REGION Network 52: MB3 Code 4037 - REGOLAZ. BORDATRICE - PASSAGGIO 04 - COMBO
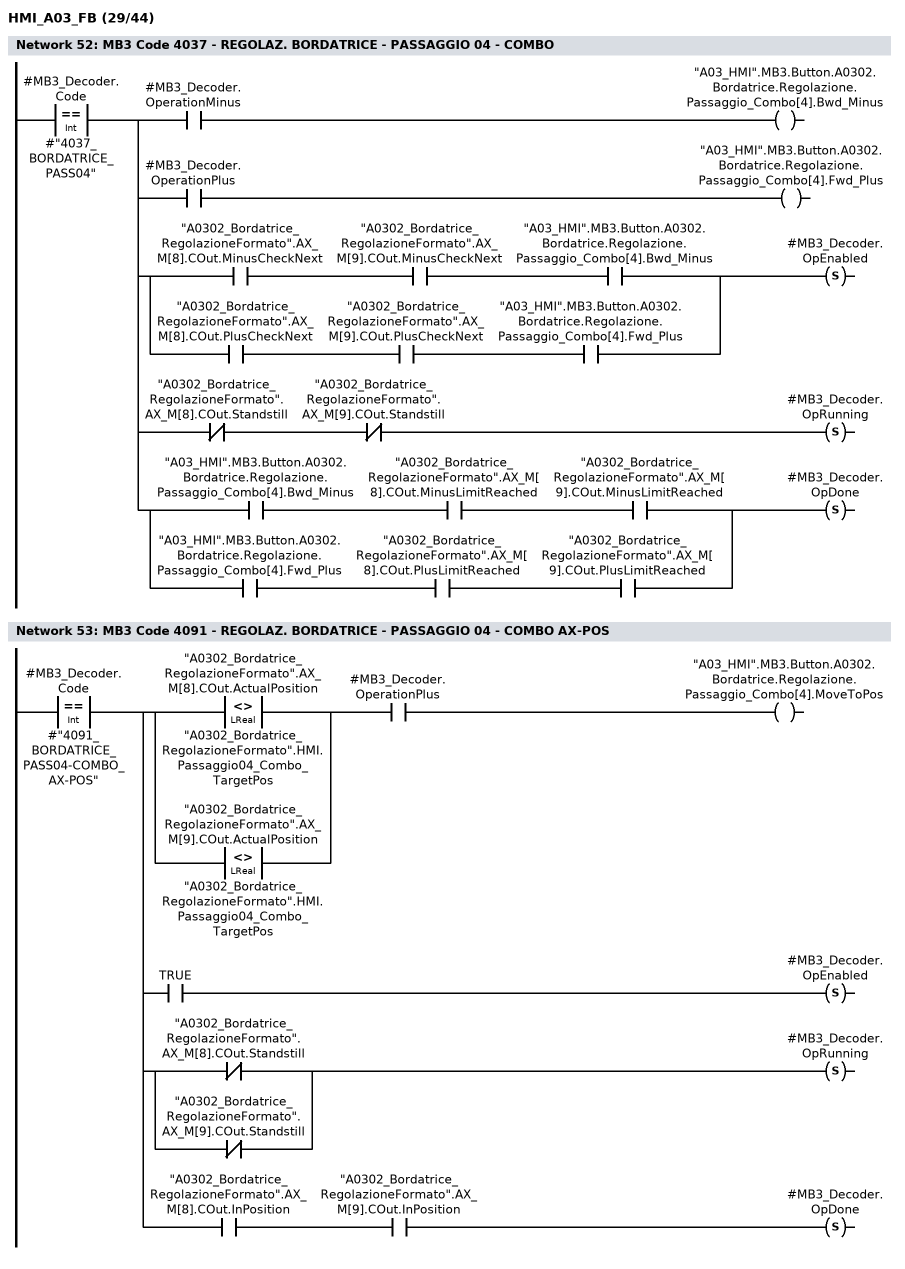
   RUNG wire#powerrail
      { S7_Templates := "SrcType := Int" } EQ_Contact(in1 := #MB3_Decoder.Code, in2 := #"4037_BORDATRICE_PASS04")
      wire#w1
      Contact( #MB3_Decoder.OperationMinus )
      Coil( "A03_HMI".MB3.Button.A0302.Bordatrice.Regolazione.Passaggio_Combo[4].Bwd_Minus )
   END_RUNG
   RUNG wire#w1
      Contact( #MB3_Decoder.OperationPlus )
      Coil( "A03_HMI".MB3.Button.A0302.Bordatrice.Regolazione.Passaggio_Combo[4].Fwd_Plus )
   END_RUNG
   RUNG wire#w1
      Contact( "A0302_Bordatrice_RegolazioneFormato".AX_M[8].COut.MinusCheckNext )
      Contact( "A0302_Bordatrice_RegolazioneFormato".AX_M[9].COut.MinusCheckNext )
      Contact( "A03_HMI".MB3.Button.A0302.Bordatrice.Regolazione.Passaggio_Combo[4].Bwd_Minus )
      wire#w2
      S_Coil( #MB3_Decoder.OpEnabled )
   END_RUNG
   RUNG wire#w1
      Contact( "A0302_Bordatrice_RegolazioneFormato".AX_M[8].COut.PlusCheckNext )
      Contact( "A0302_Bordatrice_RegolazioneFormato".AX_M[9].COut.PlusCheckNext )
      Contact( "A03_HMI".MB3.Button.A0302.Bordatrice.Regolazione.Passaggio_Combo[4].Fwd_Plus )
   END_RUNG wire#w2
   RUNG wire#w1
      I_Contact( "A0302_Bordatrice_RegolazioneFormato".AX_M[8].COut.Standstill )
      I_Contact( "A0302_Bordatrice_RegolazioneFormato".AX_M[9].COut.Standstill )
      S_Coil( #MB3_Decoder.OpRunning )
   END_RUNG
   RUNG wire#w1
      Contact( "A03_HMI".MB3.Button.A0302.Bordatrice.Regolazione.Passaggio_Combo[4].Bwd_Minus )
      Contact( "A0302_Bordatrice_RegolazioneFormato".AX_M[8].COut.MinusLimitReached )
      Contact( "A0302_Bordatrice_RegolazioneFormato".AX_M[9].COut.MinusLimitReached )
      wire#w3
      S_Coil( #MB3_Decoder.OpDone )
   END_RUNG
   RUNG wire#w1
      Contact( "A03_HMI".MB3.Button.A0302.Bordatrice.Regolazione.Passaggio_Combo[4].Fwd_Plus )
      Contact( "A0302_Bordatrice_RegolazioneFormato".AX_M[8].COut.PlusLimitReached )
      Contact( "A0302_Bordatrice_RegolazioneFormato".AX_M[9].COut.PlusLimitReached )
   END_RUNG wire#w3
   // the same network as SCL:
   #_w1 := #MB3_Decoder.Code = #"4037_BORDATRICE_PASS04";
   "A03_HMI".MB3.Button.A0302.Bordatrice.Regolazione.Passaggio_Combo[4].Bwd_Minus := #_w1 AND #MB3_Decoder.OperationMinus;
   "A03_HMI".MB3.Button.A0302.Bordatrice.Regolazione.Passaggio_Combo[4].Fwd_Plus := #_w1 AND #MB3_Decoder.OperationPlus;
   IF #_w1 AND (("A0302_Bordatrice_RegolazioneFormato".AX_M[8].COut.MinusCheckNext AND "A0302_Bordatrice_RegolazioneFormato".AX_M[9].COut.MinusCheckNext AND "A03_HMI".MB3.Button.A0302.Bordatrice.Regolazione.Passaggio_Combo[4].Bwd_Minus) OR ("A0302_Bordatrice_RegolazioneFormato".AX_M[8].COut.PlusCheckNext AND "A0302_Bordatrice_RegolazioneFormato".AX_M[9].COut.PlusCheckNext AND "A03_HMI".MB3.Button.A0302.Bordatrice.Regolazione.Passaggio_Combo[4].Fwd_Plus)) THEN
       #MB3_Decoder.OpEnabled := TRUE;
   END_IF;
   IF #_w1 AND NOT "A0302_Bordatrice_RegolazioneFormato".AX_M[8].COut.Standstill AND NOT "A0302_Bordatrice_RegolazioneFormato".AX_M[9].COut.Standstill THEN
       #MB3_Decoder.OpRunning := TRUE;
   END_IF;
   IF #_w1 AND (("A03_HMI".MB3.Button.A0302.Bordatrice.Regolazione.Passaggio_Combo[4].Bwd_Minus AND "A0302_Bordatrice_RegolazioneFormato".AX_M[8].COut.MinusLimitReached AND "A0302_Bordatrice_RegolazioneFormato".AX_M[9].COut.MinusLimitReached) OR ("A03_HMI".MB3.Button.A0302.Bordatrice.Regolazione.Passaggio_Combo[4].Fwd_Plus AND "A0302_Bordatrice_RegolazioneFormato".AX_M[8].COut.PlusLimitReached AND "A0302_Bordatrice_RegolazioneFormato".AX_M[9].COut.PlusLimitReached)) THEN
       #MB3_Decoder.OpDone := TRUE;
   END_IF;
END_REGION

REGION Network 53: MB3 Code 4091 - REGOLAZ. BORDATRICE - PASSAGGIO 04 - COMBO AX-POS
   RUNG wire#powerrail
      { S7_Templates := "SrcType := Int" } EQ_Contact(in1 := #MB3_Decoder.Code, in2 := #"4091_BORDATRICE_PASS04-COMBO_AX-POS")
      wire#w1
      { S7_Templates := "SrcType := LReal" } NE_Contact(in1 := "A0302_Bordatrice_RegolazioneFormato".AX_M[8].COut.ActualPosition, in2 := "A0302_Bordatrice_RegolazioneFormato".HMI.Passaggio04_Combo_TargetPos)
      wire#w2
      Contact( #MB3_Decoder.OperationPlus )
      Coil( "A03_HMI".MB3.Button.A0302.Bordatrice.Regolazione.Passaggio_Combo[4].MoveToPos )
   END_RUNG
   RUNG wire#w1
      { S7_Templates := "SrcType := LReal" } NE_Contact(in1 := "A0302_Bordatrice_RegolazioneFormato".AX_M[9].COut.ActualPosition, in2 := "A0302_Bordatrice_RegolazioneFormato".HMI.Passaggio04_Combo_TargetPos)
   END_RUNG wire#w2
   RUNG wire#w1
      Contact( TRUE )
      S_Coil( #MB3_Decoder.OpEnabled )
   END_RUNG
   RUNG wire#w1
      I_Contact( "A0302_Bordatrice_RegolazioneFormato".AX_M[8].COut.Standstill )
      wire#w3
      S_Coil( #MB3_Decoder.OpRunning )
   END_RUNG
   RUNG wire#w1
      I_Contact( "A0302_Bordatrice_RegolazioneFormato".AX_M[9].COut.Standstill )
   END_RUNG wire#w3
   RUNG wire#w1
      Contact( "A0302_Bordatrice_RegolazioneFormato".AX_M[8].COut.InPosition )
      Contact( "A0302_Bordatrice_RegolazioneFormato".AX_M[9].COut.InPosition )
      S_Coil( #MB3_Decoder.OpDone )
   END_RUNG
   // the same network as SCL:
   #_w1 := #MB3_Decoder.Code = #"4091_BORDATRICE_PASS04-COMBO_AX-POS";
   "A03_HMI".MB3.Button.A0302.Bordatrice.Regolazione.Passaggio_Combo[4].MoveToPos := #_w1 AND (("A0302_Bordatrice_RegolazioneFormato".AX_M[8].COut.ActualPosition <> "A0302_Bordatrice_RegolazioneFormato".HMI.Passaggio04_Combo_TargetPos) OR ("A0302_Bordatrice_RegolazioneFormato".AX_M[9].COut.ActualPosition <> "A0302_Bordatrice_RegolazioneFormato".HMI.Passaggio04_Combo_TargetPos)) AND #MB3_Decoder.OperationPlus;
   IF #_w1 AND TRUE THEN #MB3_Decoder.OpEnabled := TRUE; END_IF;
   IF #_w1 AND (NOT "A0302_Bordatrice_RegolazioneFormato".AX_M[8].COut.Standstill OR NOT "A0302_Bordatrice_RegolazioneFormato".AX_M[9].COut.Standstill) THEN
       #MB3_Decoder.OpRunning := TRUE;
   END_IF;
   IF #_w1 AND "A0302_Bordatrice_RegolazioneFormato".AX_M[8].COut.InPosition AND "A0302_Bordatrice_RegolazioneFormato".AX_M[9].COut.InPosition THEN
       #MB3_Decoder.OpDone := TRUE;
   END_IF;
END_REGION

REGION Network 54: MB3 Code 4086 - REGOLAZ. BORDATRICE - PASSAGGIO 04 - LATO-OP
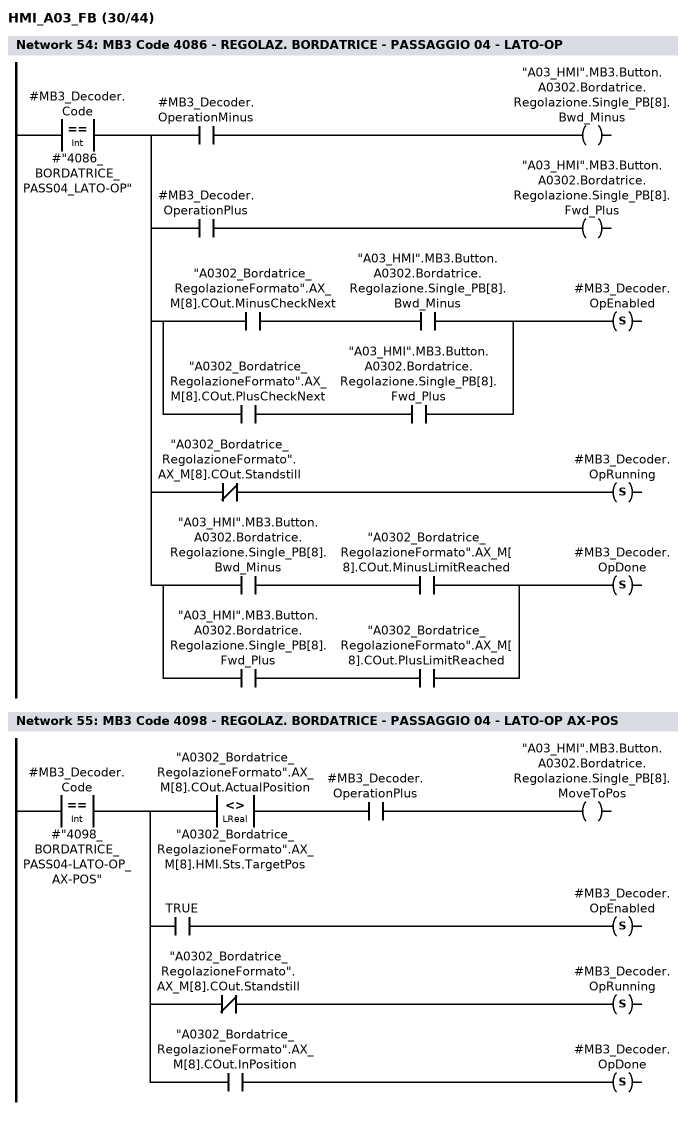
   RUNG wire#powerrail
      { S7_Templates := "SrcType := Int" } EQ_Contact(in1 := #MB3_Decoder.Code, in2 := #"4086_BORDATRICE_PASS04_LATO-OP")
      wire#w1
      Contact( #MB3_Decoder.OperationMinus )
      Coil( "A03_HMI".MB3.Button.A0302.Bordatrice.Regolazione.Single_PB[8].Bwd_Minus )
   END_RUNG
   RUNG wire#w1
      Contact( #MB3_Decoder.OperationPlus )
      Coil( "A03_HMI".MB3.Button.A0302.Bordatrice.Regolazione.Single_PB[8].Fwd_Plus )
   END_RUNG
   RUNG wire#w1
      Contact( "A0302_Bordatrice_RegolazioneFormato".AX_M[8].COut.MinusCheckNext )
      Contact( "A03_HMI".MB3.Button.A0302.Bordatrice.Regolazione.Single_PB[8].Bwd_Minus )
      wire#w2
      S_Coil( #MB3_Decoder.OpEnabled )
   END_RUNG
   RUNG wire#w1
      Contact( "A0302_Bordatrice_RegolazioneFormato".AX_M[8].COut.PlusCheckNext )
      Contact( "A03_HMI".MB3.Button.A0302.Bordatrice.Regolazione.Single_PB[8].Fwd_Plus )
   END_RUNG wire#w2
   RUNG wire#w1
      I_Contact( "A0302_Bordatrice_RegolazioneFormato".AX_M[8].COut.Standstill )
      S_Coil( #MB3_Decoder.OpRunning )
   END_RUNG
   RUNG wire#w1
      Contact( "A03_HMI".MB3.Button.A0302.Bordatrice.Regolazione.Single_PB[8].Bwd_Minus )
      Contact( "A0302_Bordatrice_RegolazioneFormato".AX_M[8].COut.MinusLimitReached )
      wire#w3
      S_Coil( #MB3_Decoder.OpDone )
   END_RUNG
   RUNG wire#w1
      Contact( "A03_HMI".MB3.Button.A0302.Bordatrice.Regolazione.Single_PB[8].Fwd_Plus )
      Contact( "A0302_Bordatrice_RegolazioneFormato".AX_M[8].COut.PlusLimitReached )
   END_RUNG wire#w3
   // the same network as SCL:
   #_w1 := #MB3_Decoder.Code = #"4086_BORDATRICE_PASS04_LATO-OP";
   "A03_HMI".MB3.Button.A0302.Bordatrice.Regolazione.Single_PB[8].Bwd_Minus := #_w1 AND #MB3_Decoder.OperationMinus;
   "A03_HMI".MB3.Button.A0302.Bordatrice.Regolazione.Single_PB[8].Fwd_Plus := #_w1 AND #MB3_Decoder.OperationPlus;
   IF #_w1 AND (("A0302_Bordatrice_RegolazioneFormato".AX_M[8].COut.MinusCheckNext AND "A03_HMI".MB3.Button.A0302.Bordatrice.Regolazione.Single_PB[8].Bwd_Minus) OR ("A0302_Bordatrice_RegolazioneFormato".AX_M[8].COut.PlusCheckNext AND "A03_HMI".MB3.Button.A0302.Bordatrice.Regolazione.Single_PB[8].Fwd_Plus)) THEN
       #MB3_Decoder.OpEnabled := TRUE;
   END_IF;
   IF #_w1 AND NOT "A0302_Bordatrice_RegolazioneFormato".AX_M[8].COut.Standstill THEN
       #MB3_Decoder.OpRunning := TRUE;
   END_IF;
   IF #_w1 AND (("A03_HMI".MB3.Button.A0302.Bordatrice.Regolazione.Single_PB[8].Bwd_Minus AND "A0302_Bordatrice_RegolazioneFormato".AX_M[8].COut.MinusLimitReached) OR ("A03_HMI".MB3.Button.A0302.Bordatrice.Regolazione.Single_PB[8].Fwd_Plus AND "A0302_Bordatrice_RegolazioneFormato".AX_M[8].COut.PlusLimitReached)) THEN
       #MB3_Decoder.OpDone := TRUE;
   END_IF;
END_REGION

REGION Network 55: MB3 Code 4098 - REGOLAZ. BORDATRICE - PASSAGGIO 04 - LATO-OP AX-POS
   RUNG wire#powerrail
      { S7_Templates := "SrcType := Int" } EQ_Contact(in1 := #MB3_Decoder.Code, in2 := #"4098_BORDATRICE_PASS04-LATO-OP_AX-POS")
      wire#w1
      { S7_Templates := "SrcType := LReal" } NE_Contact(in1 := "A0302_Bordatrice_RegolazioneFormato".AX_M[8].COut.ActualPosition, in2 := "A0302_Bordatrice_RegolazioneFormato".AX_M[8].HMI.Sts.TargetPos)
      Contact( #MB3_Decoder.OperationPlus )
      Coil( "A03_HMI".MB3.Button.A0302.Bordatrice.Regolazione.Single_PB[8].MoveToPos )
   END_RUNG
   RUNG wire#w1
      Contact( TRUE )
      S_Coil( #MB3_Decoder.OpEnabled )
   END_RUNG
   RUNG wire#w1
      I_Contact( "A0302_Bordatrice_RegolazioneFormato".AX_M[8].COut.Standstill )
      S_Coil( #MB3_Decoder.OpRunning )
   END_RUNG
   RUNG wire#w1
      Contact( "A0302_Bordatrice_RegolazioneFormato".AX_M[8].COut.InPosition )
      S_Coil( #MB3_Decoder.OpDone )
   END_RUNG
   // the same network as SCL:
   #_w1 := #MB3_Decoder.Code = #"4098_BORDATRICE_PASS04-LATO-OP_AX-POS";
   "A03_HMI".MB3.Button.A0302.Bordatrice.Regolazione.Single_PB[8].MoveToPos := #_w1 AND ("A0302_Bordatrice_RegolazioneFormato".AX_M[8].COut.ActualPosition <> "A0302_Bordatrice_RegolazioneFormato".AX_M[8].HMI.Sts.TargetPos) AND #MB3_Decoder.OperationPlus;
   IF #_w1 AND TRUE THEN #MB3_Decoder.OpEnabled := TRUE; END_IF;
   IF #_w1 AND NOT "A0302_Bordatrice_RegolazioneFormato".AX_M[8].COut.Standstill THEN
       #MB3_Decoder.OpRunning := TRUE;
   END_IF;
   IF #_w1 AND "A0302_Bordatrice_RegolazioneFormato".AX_M[8].COut.InPosition THEN
       #MB3_Decoder.OpDone := TRUE;
   END_IF;
END_REGION

REGION Network 56: MB3 Code 4087 - REGOLAZ. BORDATRICE - PASSAGGIO 04 - LATO-MOT
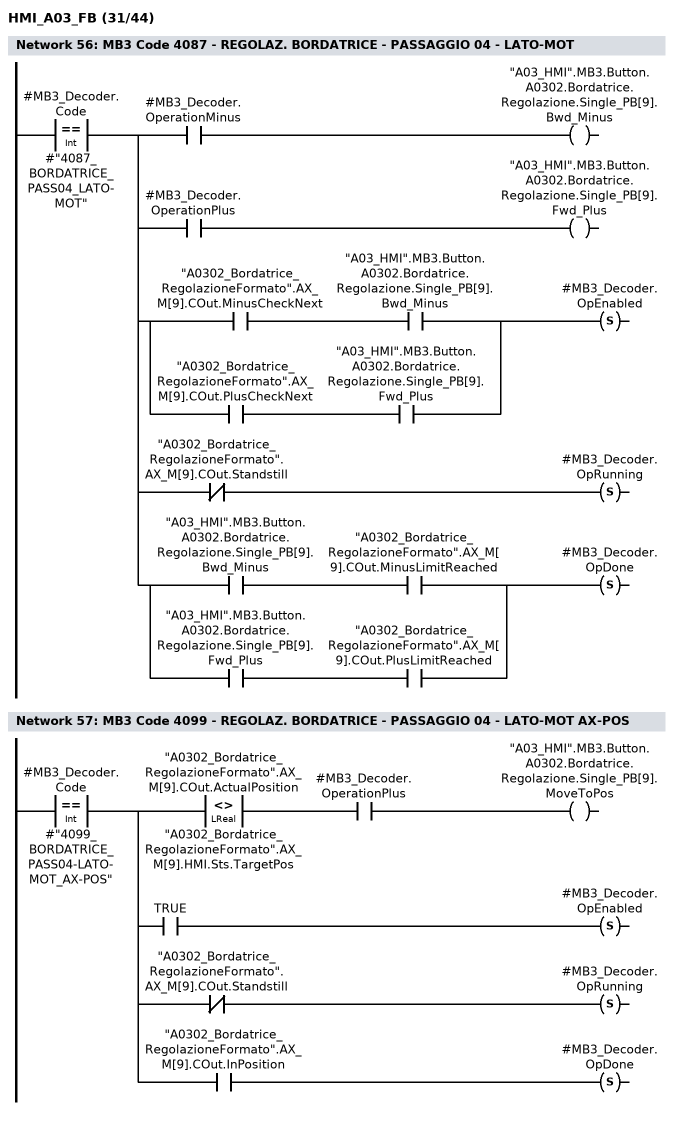
   RUNG wire#powerrail
      { S7_Templates := "SrcType := Int" } EQ_Contact(in1 := #MB3_Decoder.Code, in2 := #"4087_BORDATRICE_PASS04_LATO-MOT")
      wire#w1
      Contact( #MB3_Decoder.OperationMinus )
      Coil( "A03_HMI".MB3.Button.A0302.Bordatrice.Regolazione.Single_PB[9].Bwd_Minus )
   END_RUNG
   RUNG wire#w1
      Contact( #MB3_Decoder.OperationPlus )
      Coil( "A03_HMI".MB3.Button.A0302.Bordatrice.Regolazione.Single_PB[9].Fwd_Plus )
   END_RUNG
   RUNG wire#w1
      Contact( "A0302_Bordatrice_RegolazioneFormato".AX_M[9].COut.MinusCheckNext )
      Contact( "A03_HMI".MB3.Button.A0302.Bordatrice.Regolazione.Single_PB[9].Bwd_Minus )
      wire#w2
      S_Coil( #MB3_Decoder.OpEnabled )
   END_RUNG
   RUNG wire#w1
      Contact( "A0302_Bordatrice_RegolazioneFormato".AX_M[9].COut.PlusCheckNext )
      Contact( "A03_HMI".MB3.Button.A0302.Bordatrice.Regolazione.Single_PB[9].Fwd_Plus )
   END_RUNG wire#w2
   RUNG wire#w1
      I_Contact( "A0302_Bordatrice_RegolazioneFormato".AX_M[9].COut.Standstill )
      S_Coil( #MB3_Decoder.OpRunning )
   END_RUNG
   RUNG wire#w1
      Contact( "A03_HMI".MB3.Button.A0302.Bordatrice.Regolazione.Single_PB[9].Bwd_Minus )
      Contact( "A0302_Bordatrice_RegolazioneFormato".AX_M[9].COut.MinusLimitReached )
      wire#w3
      S_Coil( #MB3_Decoder.OpDone )
   END_RUNG
   RUNG wire#w1
      Contact( "A03_HMI".MB3.Button.A0302.Bordatrice.Regolazione.Single_PB[9].Fwd_Plus )
      Contact( "A0302_Bordatrice_RegolazioneFormato".AX_M[9].COut.PlusLimitReached )
   END_RUNG wire#w3
   // the same network as SCL:
   #_w1 := #MB3_Decoder.Code = #"4087_BORDATRICE_PASS04_LATO-MOT";
   "A03_HMI".MB3.Button.A0302.Bordatrice.Regolazione.Single_PB[9].Bwd_Minus := #_w1 AND #MB3_Decoder.OperationMinus;
   "A03_HMI".MB3.Button.A0302.Bordatrice.Regolazione.Single_PB[9].Fwd_Plus := #_w1 AND #MB3_Decoder.OperationPlus;
   IF #_w1 AND (("A0302_Bordatrice_RegolazioneFormato".AX_M[9].COut.MinusCheckNext AND "A03_HMI".MB3.Button.A0302.Bordatrice.Regolazione.Single_PB[9].Bwd_Minus) OR ("A0302_Bordatrice_RegolazioneFormato".AX_M[9].COut.PlusCheckNext AND "A03_HMI".MB3.Button.A0302.Bordatrice.Regolazione.Single_PB[9].Fwd_Plus)) THEN
       #MB3_Decoder.OpEnabled := TRUE;
   END_IF;
   IF #_w1 AND NOT "A0302_Bordatrice_RegolazioneFormato".AX_M[9].COut.Standstill THEN
       #MB3_Decoder.OpRunning := TRUE;
   END_IF;
   IF #_w1 AND (("A03_HMI".MB3.Button.A0302.Bordatrice.Regolazione.Single_PB[9].Bwd_Minus AND "A0302_Bordatrice_RegolazioneFormato".AX_M[9].COut.MinusLimitReached) OR ("A03_HMI".MB3.Button.A0302.Bordatrice.Regolazione.Single_PB[9].Fwd_Plus AND "A0302_Bordatrice_RegolazioneFormato".AX_M[9].COut.PlusLimitReached)) THEN
       #MB3_Decoder.OpDone := TRUE;
   END_IF;
END_REGION

REGION Network 57: MB3 Code 4099 - REGOLAZ. BORDATRICE - PASSAGGIO 04 - LATO-MOT AX-POS
   RUNG wire#powerrail
      { S7_Templates := "SrcType := Int" } EQ_Contact(in1 := #MB3_Decoder.Code, in2 := #"4099_BORDATRICE_PASS04-LATO-MOT_AX-POS")
      wire#w1
      { S7_Templates := "SrcType := LReal" } NE_Contact(in1 := "A0302_Bordatrice_RegolazioneFormato".AX_M[9].COut.ActualPosition, in2 := "A0302_Bordatrice_RegolazioneFormato".AX_M[9].HMI.Sts.TargetPos)
      Contact( #MB3_Decoder.OperationPlus )
      Coil( "A03_HMI".MB3.Button.A0302.Bordatrice.Regolazione.Single_PB[9].MoveToPos )
   END_RUNG
   RUNG wire#w1
      Contact( TRUE )
      S_Coil( #MB3_Decoder.OpEnabled )
   END_RUNG
   RUNG wire#w1
      I_Contact( "A0302_Bordatrice_RegolazioneFormato".AX_M[9].COut.Standstill )
      S_Coil( #MB3_Decoder.OpRunning )
   END_RUNG
   RUNG wire#w1
      Contact( "A0302_Bordatrice_RegolazioneFormato".AX_M[9].COut.InPosition )
      S_Coil( #MB3_Decoder.OpDone )
   END_RUNG
   // the same network as SCL:
   #_w1 := #MB3_Decoder.Code = #"4099_BORDATRICE_PASS04-LATO-MOT_AX-POS";
   "A03_HMI".MB3.Button.A0302.Bordatrice.Regolazione.Single_PB[9].MoveToPos := #_w1 AND ("A0302_Bordatrice_RegolazioneFormato".AX_M[9].COut.ActualPosition <> "A0302_Bordatrice_RegolazioneFormato".AX_M[9].HMI.Sts.TargetPos) AND #MB3_Decoder.OperationPlus;
   IF #_w1 AND TRUE THEN #MB3_Decoder.OpEnabled := TRUE; END_IF;
   IF #_w1 AND NOT "A0302_Bordatrice_RegolazioneFormato".AX_M[9].COut.Standstill THEN
       #MB3_Decoder.OpRunning := TRUE;
   END_IF;
   IF #_w1 AND "A0302_Bordatrice_RegolazioneFormato".AX_M[9].COut.InPosition THEN
       #MB3_Decoder.OpDone := TRUE;
   END_IF;
END_REGION

REGION Network 58: MB3 Code 4041- CENTARTORI - OP
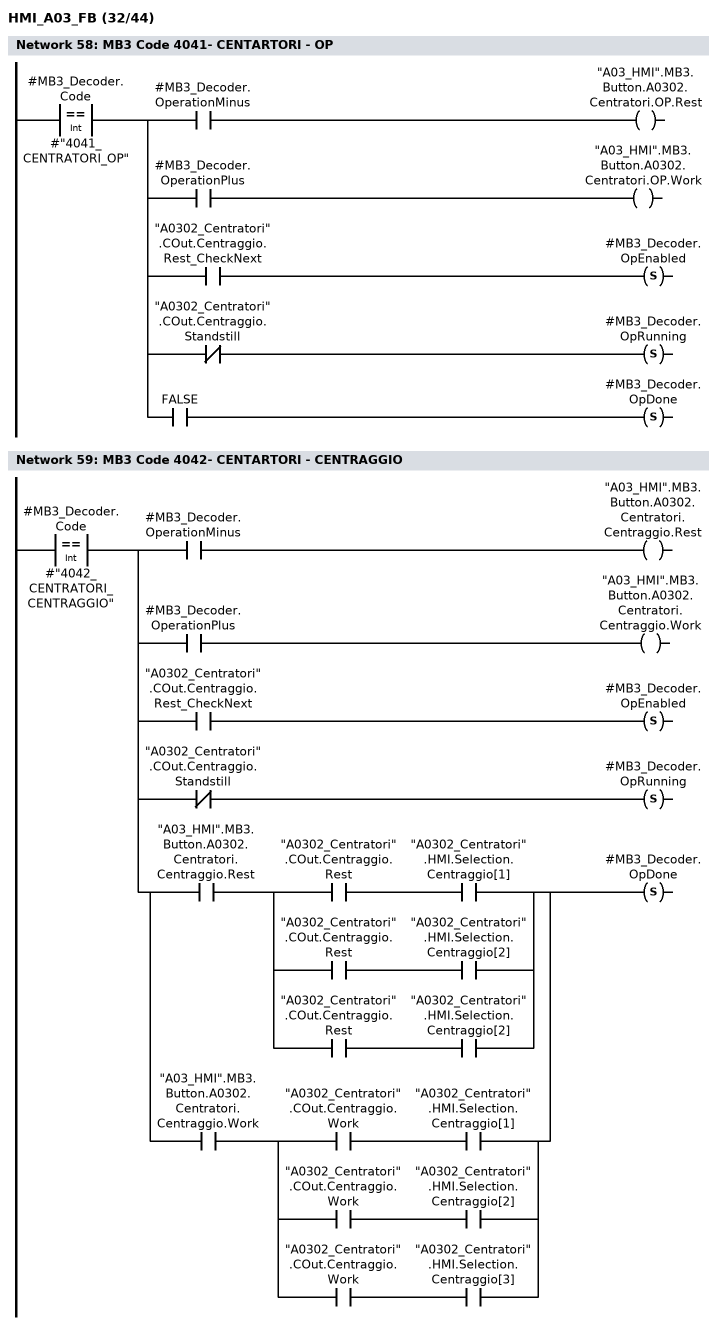
   RUNG wire#powerrail
      { S7_Templates := "SrcType := Int" } EQ_Contact(in1 := #MB3_Decoder.Code, in2 := #"4041_CENTRATORI_OP")
      wire#w1
      Contact( #MB3_Decoder.OperationMinus )
      Coil( "A03_HMI".MB3.Button.A0302.Centratori.OP.Rest )
   END_RUNG
   RUNG wire#w1
      Contact( #MB3_Decoder.OperationPlus )
      Coil( "A03_HMI".MB3.Button.A0302.Centratori.OP.Work )
   END_RUNG
   RUNG wire#w1
      Contact( "A0302_Centratori".COut.Centraggio.Rest_CheckNext )
      S_Coil( #MB3_Decoder.OpEnabled )
   END_RUNG
   RUNG wire#w1
      I_Contact( "A0302_Centratori".COut.Centraggio.Standstill )
      S_Coil( #MB3_Decoder.OpRunning )
   END_RUNG
   RUNG wire#w1
      Contact( FALSE )
      S_Coil( #MB3_Decoder.OpDone )
   END_RUNG
   // the same network as SCL:
   #_w1 := #MB3_Decoder.Code = #"4041_CENTRATORI_OP";
   "A03_HMI".MB3.Button.A0302.Centratori.OP.Rest := #_w1 AND #MB3_Decoder.OperationMinus;
   "A03_HMI".MB3.Button.A0302.Centratori.OP.Work := #_w1 AND #MB3_Decoder.OperationPlus;
   IF #_w1 AND "A0302_Centratori".COut.Centraggio.Rest_CheckNext THEN #MB3_Decoder.OpEnabled := TRUE; END_IF;
   IF #_w1 AND NOT "A0302_Centratori".COut.Centraggio.Standstill THEN #MB3_Decoder.OpRunning := TRUE; END_IF;
   IF #_w1 AND FALSE THEN #MB3_Decoder.OpDone := TRUE; END_IF;
END_REGION

REGION Network 59: MB3 Code 4042- CENTARTORI - CENTRAGGIO
   RUNG wire#powerrail
      { S7_Templates := "SrcType := Int" } EQ_Contact(in1 := #MB3_Decoder.Code, in2 := #"4042_CENTRATORI_CENTRAGGIO")
      wire#w1
      Contact( #MB3_Decoder.OperationMinus )
      Coil( "A03_HMI".MB3.Button.A0302.Centratori.Centraggio.Rest )
   END_RUNG
   RUNG wire#w1
      Contact( #MB3_Decoder.OperationPlus )
      Coil( "A03_HMI".MB3.Button.A0302.Centratori.Centraggio.Work )
   END_RUNG
   RUNG wire#w1
      Contact( "A0302_Centratori".COut.Centraggio.Rest_CheckNext )
      S_Coil( #MB3_Decoder.OpEnabled )
   END_RUNG
   RUNG wire#w1
      I_Contact( "A0302_Centratori".COut.Centraggio.Standstill )
      S_Coil( #MB3_Decoder.OpRunning )
   END_RUNG
   RUNG wire#w1
      Contact( "A03_HMI".MB3.Button.A0302.Centratori.Centraggio.Rest )
      wire#w2
      Contact( "A0302_Centratori".COut.Centraggio.Rest )
      Contact( "A0302_Centratori".HMI.Selection.Centraggio[1] )
      wire#w3
      S_Coil( #MB3_Decoder.OpDone )
   END_RUNG
   RUNG wire#w2
      Contact( "A0302_Centratori".COut.Centraggio.Rest )
      Contact( "A0302_Centratori".HMI.Selection.Centraggio[2] )
   END_RUNG wire#w3
   RUNG wire#w2
      Contact( "A0302_Centratori".COut.Centraggio.Rest )
      Contact( "A0302_Centratori".HMI.Selection.Centraggio[2] )
   END_RUNG wire#w3
   RUNG wire#w1
      Contact( "A03_HMI".MB3.Button.A0302.Centratori.Centraggio.Work )
      wire#w4
      Contact( "A0302_Centratori".COut.Centraggio.Work )
      Contact( "A0302_Centratori".HMI.Selection.Centraggio[1] )
   END_RUNG wire#w3
   RUNG wire#w4
      Contact( "A0302_Centratori".COut.Centraggio.Work )
      Contact( "A0302_Centratori".HMI.Selection.Centraggio[2] )
   END_RUNG wire#w3
   RUNG wire#w4
      Contact( "A0302_Centratori".COut.Centraggio.Work )
      Contact( "A0302_Centratori".HMI.Selection.Centraggio[3] )
   END_RUNG wire#w3
   // the same network as SCL:
   #_w1 := #MB3_Decoder.Code = #"4042_CENTRATORI_CENTRAGGIO";
   "A03_HMI".MB3.Button.A0302.Centratori.Centraggio.Rest := #_w1 AND #MB3_Decoder.OperationMinus;
   "A03_HMI".MB3.Button.A0302.Centratori.Centraggio.Work := #_w1 AND #MB3_Decoder.OperationPlus;
   IF #_w1 AND "A0302_Centratori".COut.Centraggio.Rest_CheckNext THEN #MB3_Decoder.OpEnabled := TRUE; END_IF;
   IF #_w1 AND NOT "A0302_Centratori".COut.Centraggio.Standstill THEN #MB3_Decoder.OpRunning := TRUE; END_IF;
   IF #_w1 AND (("A03_HMI".MB3.Button.A0302.Centratori.Centraggio.Rest AND (("A0302_Centratori".COut.Centraggio.Rest AND "A0302_Centratori".HMI.Selection.Centraggio[1]) OR ("A0302_Centratori".COut.Centraggio.Rest AND "A0302_Centratori".HMI.Selection.Centraggio[2]) OR ("A0302_Centratori".COut.Centraggio.Rest AND "A0302_Centratori".HMI.Selection.Centraggio[2]))) OR ("A03_HMI".MB3.Button.A0302.Centratori.Centraggio.Work AND (("A0302_Centratori".COut.Centraggio.Work AND "A0302_Centratori".HMI.Selection.Centraggio[1]) OR ("A0302_Centratori".COut.Centraggio.Work AND "A0302_Centratori".HMI.Selection.Centraggio[2]) OR ("A0302_Centratori".COut.Centraggio.Work AND "A0302_Centratori".HMI.Selection.Centraggio[3])))) THEN
       #MB3_Decoder.OpDone := TRUE;
   END_IF;
END_REGION

REGION Network 60: MB3 Code 4043- CENTARTORI - SOLLEVAMENTO
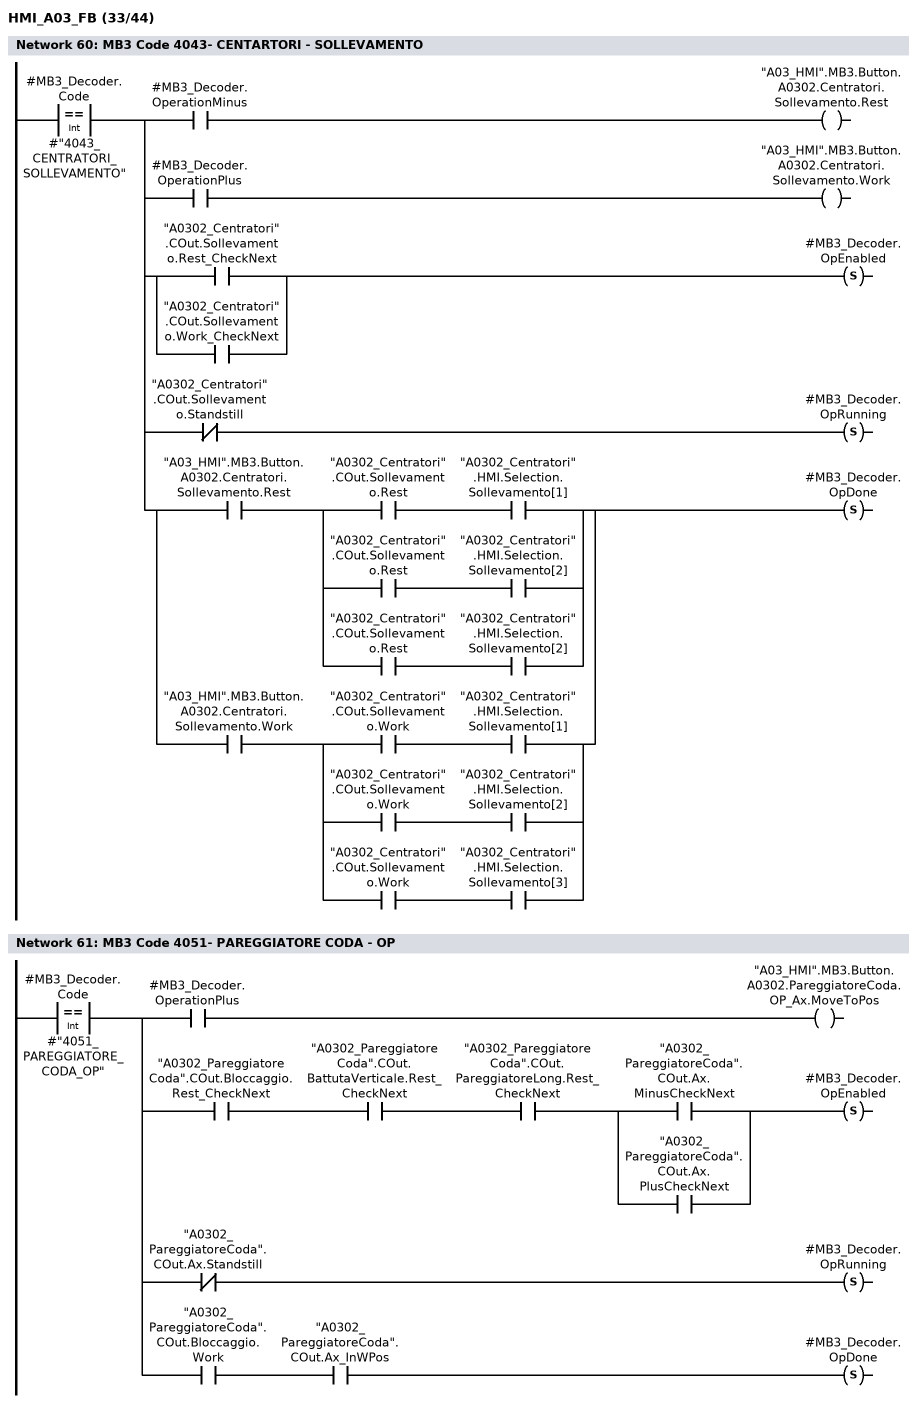
   RUNG wire#powerrail
      { S7_Templates := "SrcType := Int" } EQ_Contact(in1 := #MB3_Decoder.Code, in2 := #"4043_CENTRATORI_SOLLEVAMENTO")
      wire#w1
      Contact( #MB3_Decoder.OperationMinus )
      Coil( "A03_HMI".MB3.Button.A0302.Centratori.Sollevamento.Rest )
   END_RUNG
   RUNG wire#w1
      Contact( #MB3_Decoder.OperationPlus )
      Coil( "A03_HMI".MB3.Button.A0302.Centratori.Sollevamento.Work )
   END_RUNG
   RUNG wire#w1
      Contact( "A0302_Centratori".COut.Sollevamento.Rest_CheckNext )
      wire#w2
      S_Coil( #MB3_Decoder.OpEnabled )
   END_RUNG
   RUNG wire#w1
      Contact( "A0302_Centratori".COut.Sollevamento.Work_CheckNext )
   END_RUNG wire#w2
   RUNG wire#w1
      I_Contact( "A0302_Centratori".COut.Sollevamento.Standstill )
      S_Coil( #MB3_Decoder.OpRunning )
   END_RUNG
   RUNG wire#w1
      Contact( "A03_HMI".MB3.Button.A0302.Centratori.Sollevamento.Rest )
      wire#w3
      Contact( "A0302_Centratori".COut.Sollevamento.Rest )
      Contact( "A0302_Centratori".HMI.Selection.Sollevamento[1] )
      wire#w4
      S_Coil( #MB3_Decoder.OpDone )
   END_RUNG
   RUNG wire#w3
      Contact( "A0302_Centratori".COut.Sollevamento.Rest )
      Contact( "A0302_Centratori".HMI.Selection.Sollevamento[2] )
   END_RUNG wire#w4
   RUNG wire#w3
      Contact( "A0302_Centratori".COut.Sollevamento.Rest )
      Contact( "A0302_Centratori".HMI.Selection.Sollevamento[2] )
   END_RUNG wire#w4
   RUNG wire#w1
      Contact( "A03_HMI".MB3.Button.A0302.Centratori.Sollevamento.Work )
      wire#w5
      Contact( "A0302_Centratori".COut.Sollevamento.Work )
      Contact( "A0302_Centratori".HMI.Selection.Sollevamento[1] )
   END_RUNG wire#w4
   RUNG wire#w5
      Contact( "A0302_Centratori".COut.Sollevamento.Work )
      Contact( "A0302_Centratori".HMI.Selection.Sollevamento[2] )
   END_RUNG wire#w4
   RUNG wire#w5
      Contact( "A0302_Centratori".COut.Sollevamento.Work )
      Contact( "A0302_Centratori".HMI.Selection.Sollevamento[3] )
   END_RUNG wire#w4
   // the same network as SCL:
   #_w1 := #MB3_Decoder.Code = #"4043_CENTRATORI_SOLLEVAMENTO";
   "A03_HMI".MB3.Button.A0302.Centratori.Sollevamento.Rest := #_w1 AND #MB3_Decoder.OperationMinus;
   "A03_HMI".MB3.Button.A0302.Centratori.Sollevamento.Work := #_w1 AND #MB3_Decoder.OperationPlus;
   IF #_w1 AND ("A0302_Centratori".COut.Sollevamento.Rest_CheckNext OR "A0302_Centratori".COut.Sollevamento.Work_CheckNext) THEN
       #MB3_Decoder.OpEnabled := TRUE;
   END_IF;
   IF #_w1 AND NOT "A0302_Centratori".COut.Sollevamento.Standstill THEN
       #MB3_Decoder.OpRunning := TRUE;
   END_IF;
   IF #_w1 AND (("A03_HMI".MB3.Button.A0302.Centratori.Sollevamento.Rest AND (("A0302_Centratori".COut.Sollevamento.Rest AND "A0302_Centratori".HMI.Selection.Sollevamento[1]) OR ("A0302_Centratori".COut.Sollevamento.Rest AND "A0302_Centratori".HMI.Selection.Sollevamento[2]) OR ("A0302_Centratori".COut.Sollevamento.Rest AND "A0302_Centratori".HMI.Selection.Sollevamento[2]))) OR ("A03_HMI".MB3.Button.A0302.Centratori.Sollevamento.Work AND (("A0302_Centratori".COut.Sollevamento.Work AND "A0302_Centratori".HMI.Selection.Sollevamento[1]) OR ("A0302_Centratori".COut.Sollevamento.Work AND "A0302_Centratori".HMI.Selection.Sollevamento[2]) OR ("A0302_Centratori".COut.Sollevamento.Work AND "A0302_Centratori".HMI.Selection.Sollevamento[3])))) THEN
       #MB3_Decoder.OpDone := TRUE;
   END_IF;
END_REGION

REGION Network 61: MB3 Code 4051- PAREGGIATORE CODA - OP
   RUNG wire#powerrail
      { S7_Templates := "SrcType := Int" } EQ_Contact(in1 := #MB3_Decoder.Code, in2 := #"4051_PAREGGIATORE_CODA_OP")
      wire#w1
      Contact( #MB3_Decoder.OperationPlus )
      Coil( "A03_HMI".MB3.Button.A0302.PareggiatoreCoda.OP_Ax.MoveToPos )
   END_RUNG
   RUNG wire#w1
      Contact( "A0302_PareggiatoreCoda".COut.Bloccaggio.Rest_CheckNext )
      Contact( "A0302_PareggiatoreCoda".COut.BattutaVerticale.Rest_CheckNext )
      Contact( "A0302_PareggiatoreCoda".COut.PareggiatoreLong.Rest_CheckNext )
      wire#w2
      Contact( "A0302_PareggiatoreCoda".COut.Ax.MinusCheckNext )
      wire#w3
      S_Coil( #MB3_Decoder.OpEnabled )
   END_RUNG
   RUNG wire#w2
      Contact( "A0302_PareggiatoreCoda".COut.Ax.PlusCheckNext )
   END_RUNG wire#w3
   RUNG wire#w1
      I_Contact( "A0302_PareggiatoreCoda".COut.Ax.Standstill )
      S_Coil( #MB3_Decoder.OpRunning )
   END_RUNG
   RUNG wire#w1
      Contact( "A0302_PareggiatoreCoda".COut.Bloccaggio.Work )
      Contact( "A0302_PareggiatoreCoda".COut.Ax_InWPos )
      S_Coil( #MB3_Decoder.OpDone )
   END_RUNG
   // the same network as SCL:
   #_w1 := #MB3_Decoder.Code = #"4051_PAREGGIATORE_CODA_OP";
   "A03_HMI".MB3.Button.A0302.PareggiatoreCoda.OP_Ax.MoveToPos := #_w1 AND #MB3_Decoder.OperationPlus;
   IF #_w1 AND "A0302_PareggiatoreCoda".COut.Bloccaggio.Rest_CheckNext AND "A0302_PareggiatoreCoda".COut.BattutaVerticale.Rest_CheckNext AND "A0302_PareggiatoreCoda".COut.PareggiatoreLong.Rest_CheckNext AND ("A0302_PareggiatoreCoda".COut.Ax.MinusCheckNext OR "A0302_PareggiatoreCoda".COut.Ax.PlusCheckNext) THEN
       #MB3_Decoder.OpEnabled := TRUE;
   END_IF;
   IF #_w1 AND NOT "A0302_PareggiatoreCoda".COut.Ax.Standstill THEN #MB3_Decoder.OpRunning := TRUE; END_IF;
   IF #_w1 AND "A0302_PareggiatoreCoda".COut.Bloccaggio.Work AND "A0302_PareggiatoreCoda".COut.Ax_InWPos THEN
       #MB3_Decoder.OpDone := TRUE;
   END_IF;
END_REGION

REGION Network 62: MB3 Code 4052 - PAREGGIATORE CODA -AX
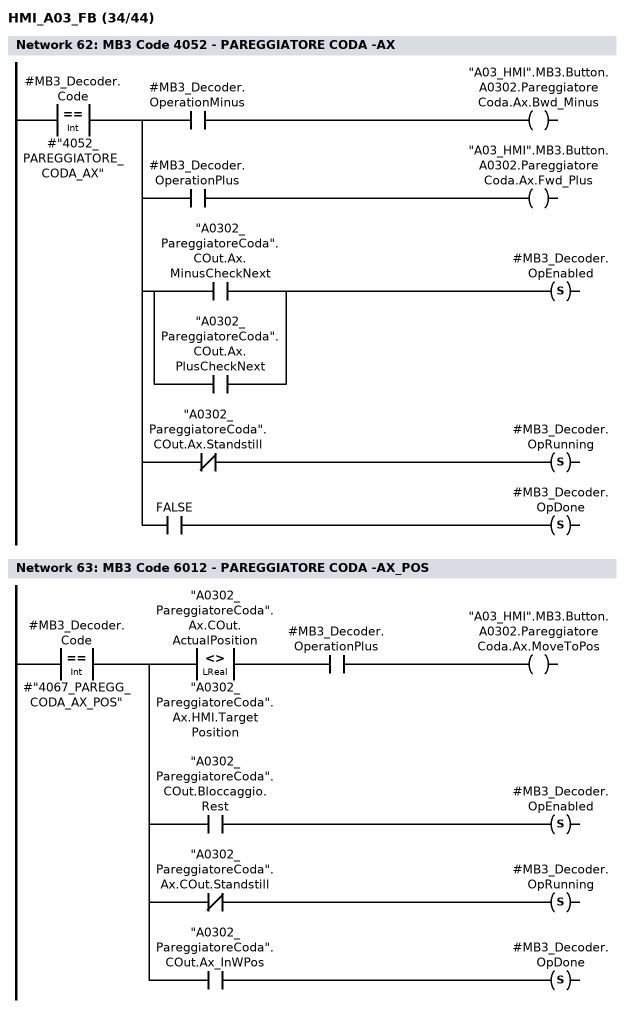
   RUNG wire#powerrail
      { S7_Templates := "SrcType := Int" } EQ_Contact(in1 := #MB3_Decoder.Code, in2 := #"4052_PAREGGIATORE_CODA_AX")
      wire#w1
      Contact( #MB3_Decoder.OperationMinus )
      Coil( "A03_HMI".MB3.Button.A0302.PareggiatoreCoda.Ax.Bwd_Minus )
   END_RUNG
   RUNG wire#w1
      Contact( #MB3_Decoder.OperationPlus )
      Coil( "A03_HMI".MB3.Button.A0302.PareggiatoreCoda.Ax.Fwd_Plus )
   END_RUNG
   RUNG wire#w1
      Contact( "A0302_PareggiatoreCoda".COut.Ax.MinusCheckNext )
      wire#w2
      S_Coil( #MB3_Decoder.OpEnabled )
   END_RUNG
   RUNG wire#w1
      Contact( "A0302_PareggiatoreCoda".COut.Ax.PlusCheckNext )
   END_RUNG wire#w2
   RUNG wire#w1
      I_Contact( "A0302_PareggiatoreCoda".COut.Ax.Standstill )
      S_Coil( #MB3_Decoder.OpRunning )
   END_RUNG
   RUNG wire#w1
      Contact( FALSE )
      S_Coil( #MB3_Decoder.OpDone )
   END_RUNG
   // the same network as SCL:
   #_w1 := #MB3_Decoder.Code = #"4052_PAREGGIATORE_CODA_AX";
   "A03_HMI".MB3.Button.A0302.PareggiatoreCoda.Ax.Bwd_Minus := #_w1 AND #MB3_Decoder.OperationMinus;
   "A03_HMI".MB3.Button.A0302.PareggiatoreCoda.Ax.Fwd_Plus := #_w1 AND #MB3_Decoder.OperationPlus;
   IF #_w1 AND ("A0302_PareggiatoreCoda".COut.Ax.MinusCheckNext OR "A0302_PareggiatoreCoda".COut.Ax.PlusCheckNext) THEN
       #MB3_Decoder.OpEnabled := TRUE;
   END_IF;
   IF #_w1 AND NOT "A0302_PareggiatoreCoda".COut.Ax.Standstill THEN #MB3_Decoder.OpRunning := TRUE; END_IF;
   IF #_w1 AND FALSE THEN #MB3_Decoder.OpDone := TRUE; END_IF;
END_REGION

REGION Network 63: MB3 Code 6012 - PAREGGIATORE CODA -AX_POS
   RUNG wire#powerrail
      { S7_Templates := "SrcType := Int" } EQ_Contact(in1 := #MB3_Decoder.Code, in2 := #"4067_PAREGG_CODA_AX_POS")
      wire#w1
      { S7_Templates := "SrcType := LReal" } NE_Contact(in1 := "A0302_PareggiatoreCoda".Ax.COut.ActualPosition, in2 := "A0302_PareggiatoreCoda".Ax.HMI.TargetPosition)
      Contact( #MB3_Decoder.OperationPlus )
      Coil( "A03_HMI".MB3.Button.A0302.PareggiatoreCoda.Ax.MoveToPos )
   END_RUNG
   RUNG wire#w1
      Contact( "A0302_PareggiatoreCoda".COut.Bloccaggio.Rest )
      S_Coil( #MB3_Decoder.OpEnabled )
   END_RUNG
   RUNG wire#w1
      I_Contact( "A0302_PareggiatoreCoda".Ax.COut.Standstill )
      S_Coil( #MB3_Decoder.OpRunning )
   END_RUNG
   RUNG wire#w1
      Contact( "A0302_PareggiatoreCoda".COut.Ax_InWPos )
      S_Coil( #MB3_Decoder.OpDone )
   END_RUNG
   // the same network as SCL:
   #_w1 := #MB3_Decoder.Code = #"4067_PAREGG_CODA_AX_POS";
   "A03_HMI".MB3.Button.A0302.PareggiatoreCoda.Ax.MoveToPos := #_w1 AND ("A0302_PareggiatoreCoda".Ax.COut.ActualPosition <> "A0302_PareggiatoreCoda".Ax.HMI.TargetPosition) AND #MB3_Decoder.OperationPlus;
   IF #_w1 AND "A0302_PareggiatoreCoda".COut.Bloccaggio.Rest THEN #MB3_Decoder.OpEnabled := TRUE; END_IF;
   IF #_w1 AND NOT "A0302_PareggiatoreCoda".Ax.COut.Standstill THEN #MB3_Decoder.OpRunning := TRUE; END_IF;
   IF #_w1 AND "A0302_PareggiatoreCoda".COut.Ax_InWPos THEN #MB3_Decoder.OpDone := TRUE; END_IF;
END_REGION

REGION Network 64: MB3 Code 4053 - PAREGGIATORE CODA - BLOCCAGGIO
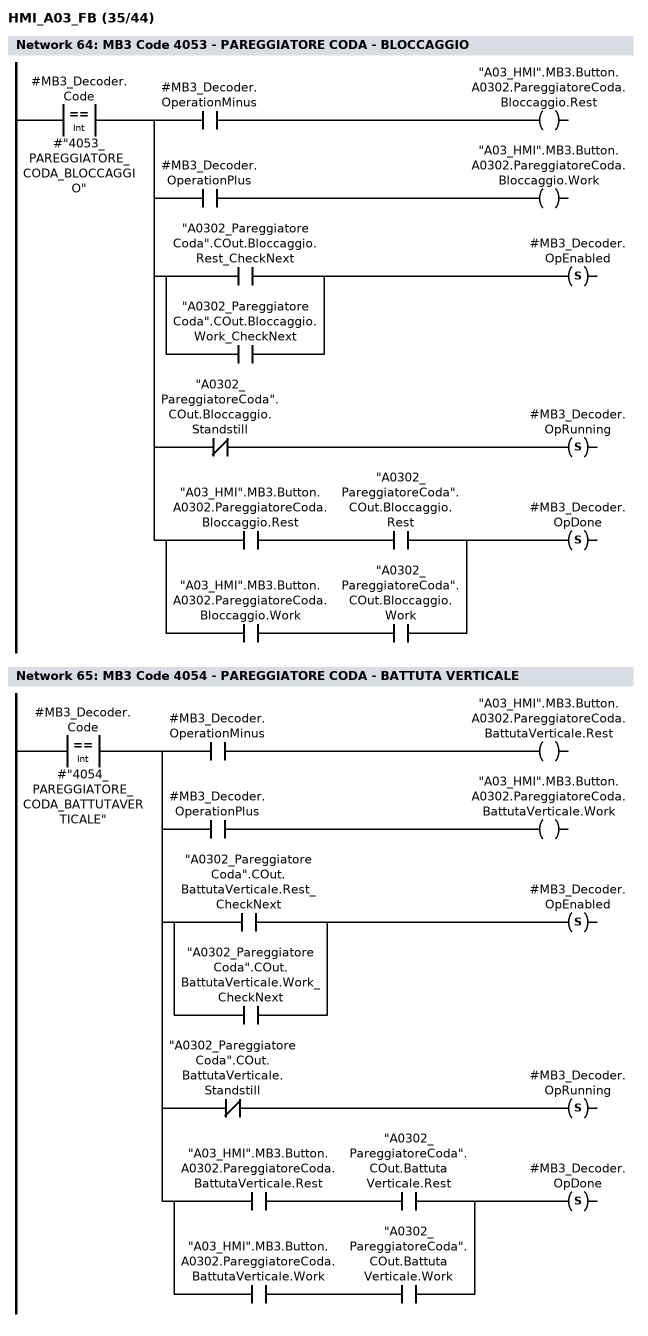
   RUNG wire#powerrail
      { S7_Templates := "SrcType := Int" } EQ_Contact(in1 := #MB3_Decoder.Code, in2 := #"4053_PAREGGIATORE_CODA_BLOCCAGGIO")
      wire#w1
      Contact( #MB3_Decoder.OperationMinus )
      Coil( "A03_HMI".MB3.Button.A0302.PareggiatoreCoda.Bloccaggio.Rest )
   END_RUNG
   RUNG wire#w1
      Contact( #MB3_Decoder.OperationPlus )
      Coil( "A03_HMI".MB3.Button.A0302.PareggiatoreCoda.Bloccaggio.Work )
   END_RUNG
   RUNG wire#w1
      Contact( "A0302_PareggiatoreCoda".COut.Bloccaggio.Rest_CheckNext )
      wire#w2
      S_Coil( #MB3_Decoder.OpEnabled )
   END_RUNG
   RUNG wire#w1
      Contact( "A0302_PareggiatoreCoda".COut.Bloccaggio.Work_CheckNext )
   END_RUNG wire#w2
   RUNG wire#w1
      I_Contact( "A0302_PareggiatoreCoda".COut.Bloccaggio.Standstill )
      S_Coil( #MB3_Decoder.OpRunning )
   END_RUNG
   RUNG wire#w1
      Contact( "A03_HMI".MB3.Button.A0302.PareggiatoreCoda.Bloccaggio.Rest )
      Contact( "A0302_PareggiatoreCoda".COut.Bloccaggio.Rest )
      wire#w3
      S_Coil( #MB3_Decoder.OpDone )
   END_RUNG
   RUNG wire#w1
      Contact( "A03_HMI".MB3.Button.A0302.PareggiatoreCoda.Bloccaggio.Work )
      Contact( "A0302_PareggiatoreCoda".COut.Bloccaggio.Work )
   END_RUNG wire#w3
   // the same network as SCL:
   #_w1 := #MB3_Decoder.Code = #"4053_PAREGGIATORE_CODA_BLOCCAGGIO";
   "A03_HMI".MB3.Button.A0302.PareggiatoreCoda.Bloccaggio.Rest := #_w1 AND #MB3_Decoder.OperationMinus;
   "A03_HMI".MB3.Button.A0302.PareggiatoreCoda.Bloccaggio.Work := #_w1 AND #MB3_Decoder.OperationPlus;
   IF #_w1 AND ("A0302_PareggiatoreCoda".COut.Bloccaggio.Rest_CheckNext OR "A0302_PareggiatoreCoda".COut.Bloccaggio.Work_CheckNext) THEN
       #MB3_Decoder.OpEnabled := TRUE;
   END_IF;
   IF #_w1 AND NOT "A0302_PareggiatoreCoda".COut.Bloccaggio.Standstill THEN
       #MB3_Decoder.OpRunning := TRUE;
   END_IF;
   IF #_w1 AND (("A03_HMI".MB3.Button.A0302.PareggiatoreCoda.Bloccaggio.Rest AND "A0302_PareggiatoreCoda".COut.Bloccaggio.Rest) OR ("A03_HMI".MB3.Button.A0302.PareggiatoreCoda.Bloccaggio.Work AND "A0302_PareggiatoreCoda".COut.Bloccaggio.Work)) THEN
       #MB3_Decoder.OpDone := TRUE;
   END_IF;
END_REGION

REGION Network 65: MB3 Code 4054 - PAREGGIATORE CODA - BATTUTA VERTICALE
   RUNG wire#powerrail
      { S7_Templates := "SrcType := Int" } EQ_Contact(in1 := #MB3_Decoder.Code, in2 := #"4054_PAREGGIATORE_CODA_BATTUTAVERTICALE")
      wire#w1
      Contact( #MB3_Decoder.OperationMinus )
      Coil( "A03_HMI".MB3.Button.A0302.PareggiatoreCoda.BattutaVerticale.Rest )
   END_RUNG
   RUNG wire#w1
      Contact( #MB3_Decoder.OperationPlus )
      Coil( "A03_HMI".MB3.Button.A0302.PareggiatoreCoda.BattutaVerticale.Work )
   END_RUNG
   RUNG wire#w1
      Contact( "A0302_PareggiatoreCoda".COut.BattutaVerticale.Rest_CheckNext )
      wire#w2
      S_Coil( #MB3_Decoder.OpEnabled )
   END_RUNG
   RUNG wire#w1
      Contact( "A0302_PareggiatoreCoda".COut.BattutaVerticale.Work_CheckNext )
   END_RUNG wire#w2
   RUNG wire#w1
      I_Contact( "A0302_PareggiatoreCoda".COut.BattutaVerticale.Standstill )
      S_Coil( #MB3_Decoder.OpRunning )
   END_RUNG
   RUNG wire#w1
      Contact( "A03_HMI".MB3.Button.A0302.PareggiatoreCoda.BattutaVerticale.Rest )
      Contact( "A0302_PareggiatoreCoda".COut.BattutaVerticale.Rest )
      wire#w3
      S_Coil( #MB3_Decoder.OpDone )
   END_RUNG
   RUNG wire#w1
      Contact( "A03_HMI".MB3.Button.A0302.PareggiatoreCoda.BattutaVerticale.Work )
      Contact( "A0302_PareggiatoreCoda".COut.BattutaVerticale.Work )
   END_RUNG wire#w3
   // the same network as SCL:
   #_w1 := #MB3_Decoder.Code = #"4054_PAREGGIATORE_CODA_BATTUTAVERTICALE";
   "A03_HMI".MB3.Button.A0302.PareggiatoreCoda.BattutaVerticale.Rest := #_w1 AND #MB3_Decoder.OperationMinus;
   "A03_HMI".MB3.Button.A0302.PareggiatoreCoda.BattutaVerticale.Work := #_w1 AND #MB3_Decoder.OperationPlus;
   IF #_w1 AND ("A0302_PareggiatoreCoda".COut.BattutaVerticale.Rest_CheckNext OR "A0302_PareggiatoreCoda".COut.BattutaVerticale.Work_CheckNext) THEN
       #MB3_Decoder.OpEnabled := TRUE;
   END_IF;
   IF #_w1 AND NOT "A0302_PareggiatoreCoda".COut.BattutaVerticale.Standstill THEN
       #MB3_Decoder.OpRunning := TRUE;
   END_IF;
   IF #_w1 AND (("A03_HMI".MB3.Button.A0302.PareggiatoreCoda.BattutaVerticale.Rest AND "A0302_PareggiatoreCoda".COut.BattutaVerticale.Rest) OR ("A03_HMI".MB3.Button.A0302.PareggiatoreCoda.BattutaVerticale.Work AND "A0302_PareggiatoreCoda".COut.BattutaVerticale.Work)) THEN
       #MB3_Decoder.OpDone := TRUE;
   END_IF;
END_REGION

REGION Network 66: MB3 Code 4055 - PAREGGIATORE CODA - PAREGGIATORE LONGITUDINALE
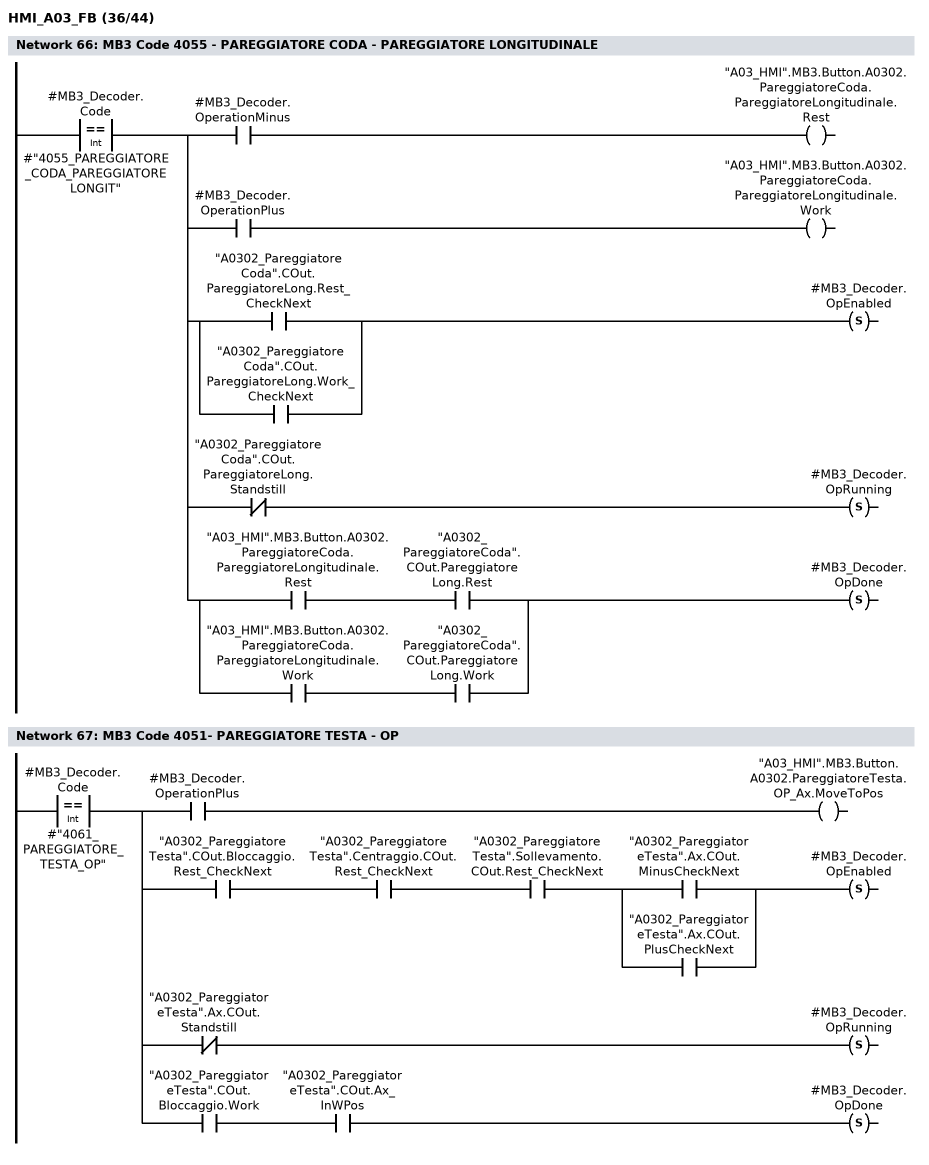
   RUNG wire#powerrail
      { S7_Templates := "SrcType := Int" } EQ_Contact(in1 := #MB3_Decoder.Code, in2 := #"4055_PAREGGIATORE_CODA_PAREGGIATORELONGIT")
      wire#w1
      Contact( #MB3_Decoder.OperationMinus )
      Coil( "A03_HMI".MB3.Button.A0302.PareggiatoreCoda.PareggiatoreLongitudinale.Rest )
   END_RUNG
   RUNG wire#w1
      Contact( #MB3_Decoder.OperationPlus )
      Coil( "A03_HMI".MB3.Button.A0302.PareggiatoreCoda.PareggiatoreLongitudinale.Work )
   END_RUNG
   RUNG wire#w1
      Contact( "A0302_PareggiatoreCoda".COut.PareggiatoreLong.Rest_CheckNext )
      wire#w2
      S_Coil( #MB3_Decoder.OpEnabled )
   END_RUNG
   RUNG wire#w1
      Contact( "A0302_PareggiatoreCoda".COut.PareggiatoreLong.Work_CheckNext )
   END_RUNG wire#w2
   RUNG wire#w1
      I_Contact( "A0302_PareggiatoreCoda".COut.PareggiatoreLong.Standstill )
      S_Coil( #MB3_Decoder.OpRunning )
   END_RUNG
   RUNG wire#w1
      Contact( "A03_HMI".MB3.Button.A0302.PareggiatoreCoda.PareggiatoreLongitudinale.Rest )
      Contact( "A0302_PareggiatoreCoda".COut.PareggiatoreLong.Rest )
      wire#w3
      S_Coil( #MB3_Decoder.OpDone )
   END_RUNG
   RUNG wire#w1
      Contact( "A03_HMI".MB3.Button.A0302.PareggiatoreCoda.PareggiatoreLongitudinale.Work )
      Contact( "A0302_PareggiatoreCoda".COut.PareggiatoreLong.Work )
   END_RUNG wire#w3
   // the same network as SCL:
   #_w1 := #MB3_Decoder.Code = #"4055_PAREGGIATORE_CODA_PAREGGIATORELONGIT";
   "A03_HMI".MB3.Button.A0302.PareggiatoreCoda.PareggiatoreLongitudinale.Rest := #_w1 AND #MB3_Decoder.OperationMinus;
   "A03_HMI".MB3.Button.A0302.PareggiatoreCoda.PareggiatoreLongitudinale.Work := #_w1 AND #MB3_Decoder.OperationPlus;
   IF #_w1 AND ("A0302_PareggiatoreCoda".COut.PareggiatoreLong.Rest_CheckNext OR "A0302_PareggiatoreCoda".COut.PareggiatoreLong.Work_CheckNext) THEN
       #MB3_Decoder.OpEnabled := TRUE;
   END_IF;
   IF #_w1 AND NOT "A0302_PareggiatoreCoda".COut.PareggiatoreLong.Standstill THEN
       #MB3_Decoder.OpRunning := TRUE;
   END_IF;
   IF #_w1 AND (("A03_HMI".MB3.Button.A0302.PareggiatoreCoda.PareggiatoreLongitudinale.Rest AND "A0302_PareggiatoreCoda".COut.PareggiatoreLong.Rest) OR ("A03_HMI".MB3.Button.A0302.PareggiatoreCoda.PareggiatoreLongitudinale.Work AND "A0302_PareggiatoreCoda".COut.PareggiatoreLong.Work)) THEN
       #MB3_Decoder.OpDone := TRUE;
   END_IF;
END_REGION

REGION Network 67: MB3 Code 4051- PAREGGIATORE TESTA - OP
   RUNG wire#powerrail
      { S7_Templates := "SrcType := Int" } EQ_Contact(in1 := #MB3_Decoder.Code, in2 := #"4061_PAREGGIATORE_TESTA_OP")
      wire#w1
      Contact( #MB3_Decoder.OperationPlus )
      Coil( "A03_HMI".MB3.Button.A0302.PareggiatoreTesta.OP_Ax.MoveToPos )
   END_RUNG
   RUNG wire#w1
      Contact( "A0302_PareggiatoreTesta".COut.Bloccaggio.Rest_CheckNext )
      Contact( "A0302_PareggiatoreTesta".Centraggio.COut.Rest_CheckNext )
      Contact( "A0302_PareggiatoreTesta".Sollevamento.COut.Rest_CheckNext )
      wire#w2
      Contact( "A0302_PareggiatoreTesta".Ax.COut.MinusCheckNext )
      wire#w3
      S_Coil( #MB3_Decoder.OpEnabled )
   END_RUNG
   RUNG wire#w2
      Contact( "A0302_PareggiatoreTesta".Ax.COut.PlusCheckNext )
   END_RUNG wire#w3
   RUNG wire#w1
      I_Contact( "A0302_PareggiatoreTesta".Ax.COut.Standstill )
      S_Coil( #MB3_Decoder.OpRunning )
   END_RUNG
   RUNG wire#w1
      Contact( "A0302_PareggiatoreTesta".COut.Bloccaggio.Work )
      Contact( "A0302_PareggiatoreTesta".COut.Ax_InWPos )
      S_Coil( #MB3_Decoder.OpDone )
   END_RUNG
   // the same network as SCL:
   #_w1 := #MB3_Decoder.Code = #"4061_PAREGGIATORE_TESTA_OP";
   "A03_HMI".MB3.Button.A0302.PareggiatoreTesta.OP_Ax.MoveToPos := #_w1 AND #MB3_Decoder.OperationPlus;
   IF #_w1 AND "A0302_PareggiatoreTesta".COut.Bloccaggio.Rest_CheckNext AND "A0302_PareggiatoreTesta".Centraggio.COut.Rest_CheckNext AND "A0302_PareggiatoreTesta".Sollevamento.COut.Rest_CheckNext AND ("A0302_PareggiatoreTesta".Ax.COut.MinusCheckNext OR "A0302_PareggiatoreTesta".Ax.COut.PlusCheckNext) THEN
       #MB3_Decoder.OpEnabled := TRUE;
   END_IF;
   IF #_w1 AND NOT "A0302_PareggiatoreTesta".Ax.COut.Standstill THEN #MB3_Decoder.OpRunning := TRUE; END_IF;
   IF #_w1 AND "A0302_PareggiatoreTesta".COut.Bloccaggio.Work AND "A0302_PareggiatoreTesta".COut.Ax_InWPos THEN
       #MB3_Decoder.OpDone := TRUE;
   END_IF;
END_REGION

REGION Network 68: MB3 Code 4062 - PAREGGIATORE TESTA -AX
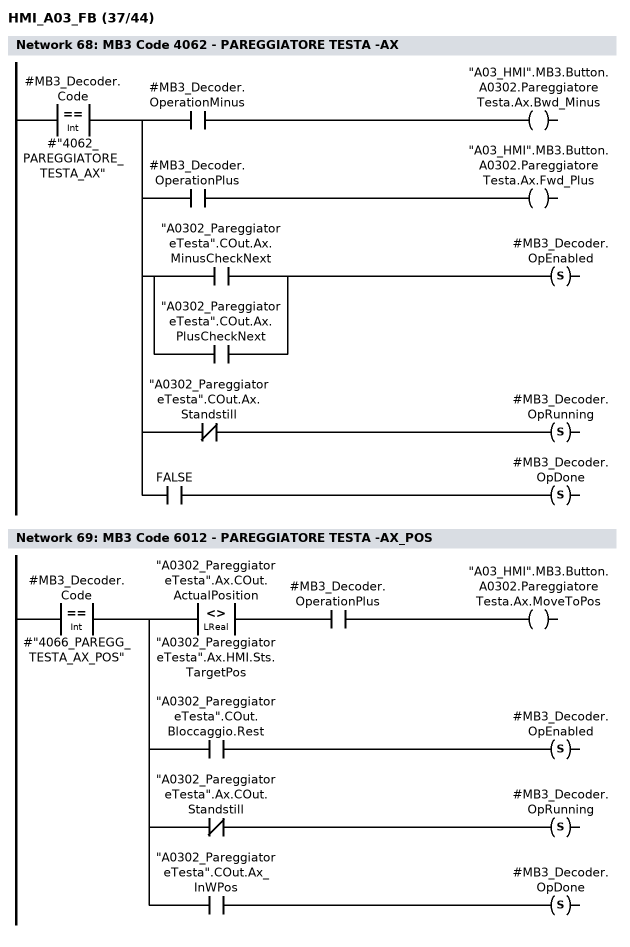
   RUNG wire#powerrail
      { S7_Templates := "SrcType := Int" } EQ_Contact(in1 := #MB3_Decoder.Code, in2 := #"4062_PAREGGIATORE_TESTA_AX")
      wire#w1
      Contact( #MB3_Decoder.OperationMinus )
      Coil( "A03_HMI".MB3.Button.A0302.PareggiatoreTesta.Ax.Bwd_Minus )
   END_RUNG
   RUNG wire#w1
      Contact( #MB3_Decoder.OperationPlus )
      Coil( "A03_HMI".MB3.Button.A0302.PareggiatoreTesta.Ax.Fwd_Plus )
   END_RUNG
   RUNG wire#w1
      Contact( "A0302_PareggiatoreTesta".COut.Ax.MinusCheckNext )
      wire#w2
      S_Coil( #MB3_Decoder.OpEnabled )
   END_RUNG
   RUNG wire#w1
      Contact( "A0302_PareggiatoreTesta".COut.Ax.PlusCheckNext )
   END_RUNG wire#w2
   RUNG wire#w1
      I_Contact( "A0302_PareggiatoreTesta".COut.Ax.Standstill )
      S_Coil( #MB3_Decoder.OpRunning )
   END_RUNG
   RUNG wire#w1
      Contact( FALSE )
      S_Coil( #MB3_Decoder.OpDone )
   END_RUNG
   // the same network as SCL:
   #_w1 := #MB3_Decoder.Code = #"4062_PAREGGIATORE_TESTA_AX";
   "A03_HMI".MB3.Button.A0302.PareggiatoreTesta.Ax.Bwd_Minus := #_w1 AND #MB3_Decoder.OperationMinus;
   "A03_HMI".MB3.Button.A0302.PareggiatoreTesta.Ax.Fwd_Plus := #_w1 AND #MB3_Decoder.OperationPlus;
   IF #_w1 AND ("A0302_PareggiatoreTesta".COut.Ax.MinusCheckNext OR "A0302_PareggiatoreTesta".COut.Ax.PlusCheckNext) THEN
       #MB3_Decoder.OpEnabled := TRUE;
   END_IF;
   IF #_w1 AND NOT "A0302_PareggiatoreTesta".COut.Ax.Standstill THEN #MB3_Decoder.OpRunning := TRUE; END_IF;
   IF #_w1 AND FALSE THEN #MB3_Decoder.OpDone := TRUE; END_IF;
END_REGION

REGION Network 69: MB3 Code 6012 - PAREGGIATORE TESTA -AX_POS
   RUNG wire#powerrail
      { S7_Templates := "SrcType := Int" } EQ_Contact(in1 := #MB3_Decoder.Code, in2 := #"4066_PAREGG_TESTA_AX_POS")
      wire#w1
      { S7_Templates := "SrcType := LReal" } NE_Contact(in1 := "A0302_PareggiatoreTesta".Ax.COut.ActualPosition, in2 := "A0302_PareggiatoreTesta".Ax.HMI.Sts.TargetPos)
      Contact( #MB3_Decoder.OperationPlus )
      Coil( "A03_HMI".MB3.Button.A0302.PareggiatoreTesta.Ax.MoveToPos )
   END_RUNG
   RUNG wire#w1
      Contact( "A0302_PareggiatoreTesta".COut.Bloccaggio.Rest )
      S_Coil( #MB3_Decoder.OpEnabled )
   END_RUNG
   RUNG wire#w1
      I_Contact( "A0302_PareggiatoreTesta".Ax.COut.Standstill )
      S_Coil( #MB3_Decoder.OpRunning )
   END_RUNG
   RUNG wire#w1
      Contact( "A0302_PareggiatoreTesta".COut.Ax_InWPos )
      S_Coil( #MB3_Decoder.OpDone )
   END_RUNG
   // the same network as SCL:
   #_w1 := #MB3_Decoder.Code = #"4066_PAREGG_TESTA_AX_POS";
   "A03_HMI".MB3.Button.A0302.PareggiatoreTesta.Ax.MoveToPos := #_w1 AND ("A0302_PareggiatoreTesta".Ax.COut.ActualPosition <> "A0302_PareggiatoreTesta".Ax.HMI.Sts.TargetPos) AND #MB3_Decoder.OperationPlus;
   IF #_w1 AND "A0302_PareggiatoreTesta".COut.Bloccaggio.Rest THEN #MB3_Decoder.OpEnabled := TRUE; END_IF;
   IF #_w1 AND NOT "A0302_PareggiatoreTesta".Ax.COut.Standstill THEN #MB3_Decoder.OpRunning := TRUE; END_IF;
   IF #_w1 AND "A0302_PareggiatoreTesta".COut.Ax_InWPos THEN #MB3_Decoder.OpDone := TRUE; END_IF;
END_REGION

REGION Network 70: MB3 Code 4063 - PAREGGIATORE TESTA - BLOCCAGGIO
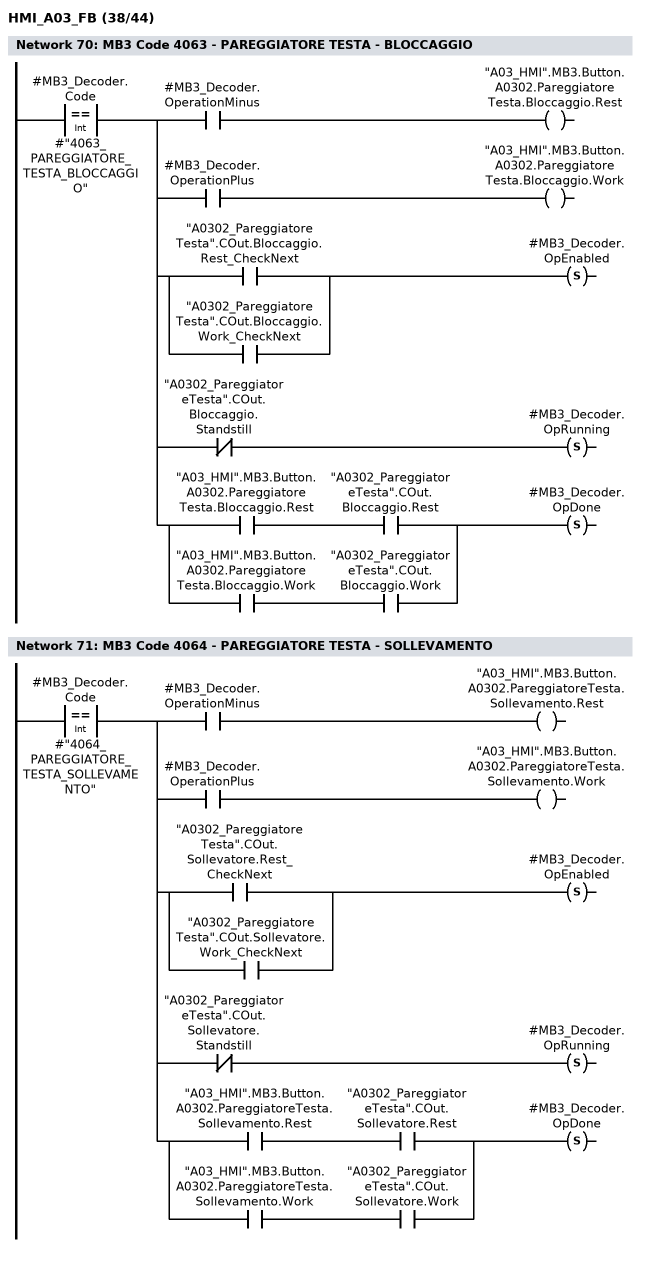
   RUNG wire#powerrail
      { S7_Templates := "SrcType := Int" } EQ_Contact(in1 := #MB3_Decoder.Code, in2 := #"4063_PAREGGIATORE_TESTA_BLOCCAGGIO")
      wire#w1
      Contact( #MB3_Decoder.OperationMinus )
      Coil( "A03_HMI".MB3.Button.A0302.PareggiatoreTesta.Bloccaggio.Rest )
   END_RUNG
   RUNG wire#w1
      Contact( #MB3_Decoder.OperationPlus )
      Coil( "A03_HMI".MB3.Button.A0302.PareggiatoreTesta.Bloccaggio.Work )
   END_RUNG
   RUNG wire#w1
      Contact( "A0302_PareggiatoreTesta".COut.Bloccaggio.Rest_CheckNext )
      wire#w2
      S_Coil( #MB3_Decoder.OpEnabled )
   END_RUNG
   RUNG wire#w1
      Contact( "A0302_PareggiatoreTesta".COut.Bloccaggio.Work_CheckNext )
   END_RUNG wire#w2
   RUNG wire#w1
      I_Contact( "A0302_PareggiatoreTesta".COut.Bloccaggio.Standstill )
      S_Coil( #MB3_Decoder.OpRunning )
   END_RUNG
   RUNG wire#w1
      Contact( "A03_HMI".MB3.Button.A0302.PareggiatoreTesta.Bloccaggio.Rest )
      Contact( "A0302_PareggiatoreTesta".COut.Bloccaggio.Rest )
      wire#w3
      S_Coil( #MB3_Decoder.OpDone )
   END_RUNG
   RUNG wire#w1
      Contact( "A03_HMI".MB3.Button.A0302.PareggiatoreTesta.Bloccaggio.Work )
      Contact( "A0302_PareggiatoreTesta".COut.Bloccaggio.Work )
   END_RUNG wire#w3
   // the same network as SCL:
   #_w1 := #MB3_Decoder.Code = #"4063_PAREGGIATORE_TESTA_BLOCCAGGIO";
   "A03_HMI".MB3.Button.A0302.PareggiatoreTesta.Bloccaggio.Rest := #_w1 AND #MB3_Decoder.OperationMinus;
   "A03_HMI".MB3.Button.A0302.PareggiatoreTesta.Bloccaggio.Work := #_w1 AND #MB3_Decoder.OperationPlus;
   IF #_w1 AND ("A0302_PareggiatoreTesta".COut.Bloccaggio.Rest_CheckNext OR "A0302_PareggiatoreTesta".COut.Bloccaggio.Work_CheckNext) THEN
       #MB3_Decoder.OpEnabled := TRUE;
   END_IF;
   IF #_w1 AND NOT "A0302_PareggiatoreTesta".COut.Bloccaggio.Standstill THEN
       #MB3_Decoder.OpRunning := TRUE;
   END_IF;
   IF #_w1 AND (("A03_HMI".MB3.Button.A0302.PareggiatoreTesta.Bloccaggio.Rest AND "A0302_PareggiatoreTesta".COut.Bloccaggio.Rest) OR ("A03_HMI".MB3.Button.A0302.PareggiatoreTesta.Bloccaggio.Work AND "A0302_PareggiatoreTesta".COut.Bloccaggio.Work)) THEN
       #MB3_Decoder.OpDone := TRUE;
   END_IF;
END_REGION

REGION Network 71: MB3 Code 4064 - PAREGGIATORE TESTA - SOLLEVAMENTO
   RUNG wire#powerrail
      { S7_Templates := "SrcType := Int" } EQ_Contact(in1 := #MB3_Decoder.Code, in2 := #"4064_PAREGGIATORE_TESTA_SOLLEVAMENTO")
      wire#w1
      Contact( #MB3_Decoder.OperationMinus )
      Coil( "A03_HMI".MB3.Button.A0302.PareggiatoreTesta.Sollevamento.Rest )
   END_RUNG
   RUNG wire#w1
      Contact( #MB3_Decoder.OperationPlus )
      Coil( "A03_HMI".MB3.Button.A0302.PareggiatoreTesta.Sollevamento.Work )
   END_RUNG
   RUNG wire#w1
      Contact( "A0302_PareggiatoreTesta".COut.Sollevatore.Rest_CheckNext )
      wire#w2
      S_Coil( #MB3_Decoder.OpEnabled )
   END_RUNG
   RUNG wire#w1
      Contact( "A0302_PareggiatoreTesta".COut.Sollevatore.Work_CheckNext )
   END_RUNG wire#w2
   RUNG wire#w1
      I_Contact( "A0302_PareggiatoreTesta".COut.Sollevatore.Standstill )
      S_Coil( #MB3_Decoder.OpRunning )
   END_RUNG
   RUNG wire#w1
      Contact( "A03_HMI".MB3.Button.A0302.PareggiatoreTesta.Sollevamento.Rest )
      Contact( "A0302_PareggiatoreTesta".COut.Sollevatore.Rest )
      wire#w3
      S_Coil( #MB3_Decoder.OpDone )
   END_RUNG
   RUNG wire#w1
      Contact( "A03_HMI".MB3.Button.A0302.PareggiatoreTesta.Sollevamento.Work )
      Contact( "A0302_PareggiatoreTesta".COut.Sollevatore.Work )
   END_RUNG wire#w3
   // the same network as SCL:
   #_w1 := #MB3_Decoder.Code = #"4064_PAREGGIATORE_TESTA_SOLLEVAMENTO";
   "A03_HMI".MB3.Button.A0302.PareggiatoreTesta.Sollevamento.Rest := #_w1 AND #MB3_Decoder.OperationMinus;
   "A03_HMI".MB3.Button.A0302.PareggiatoreTesta.Sollevamento.Work := #_w1 AND #MB3_Decoder.OperationPlus;
   IF #_w1 AND ("A0302_PareggiatoreTesta".COut.Sollevatore.Rest_CheckNext OR "A0302_PareggiatoreTesta".COut.Sollevatore.Work_CheckNext) THEN
       #MB3_Decoder.OpEnabled := TRUE;
   END_IF;
   IF #_w1 AND NOT "A0302_PareggiatoreTesta".COut.Sollevatore.Standstill THEN
       #MB3_Decoder.OpRunning := TRUE;
   END_IF;
   IF #_w1 AND (("A03_HMI".MB3.Button.A0302.PareggiatoreTesta.Sollevamento.Rest AND "A0302_PareggiatoreTesta".COut.Sollevatore.Rest) OR ("A03_HMI".MB3.Button.A0302.PareggiatoreTesta.Sollevamento.Work AND "A0302_PareggiatoreTesta".COut.Sollevatore.Work)) THEN
       #MB3_Decoder.OpDone := TRUE;
   END_IF;
END_REGION

REGION Network 72: MB3 Code 4064 - PAREGGIATORE TESTA - CENTRAGGIO
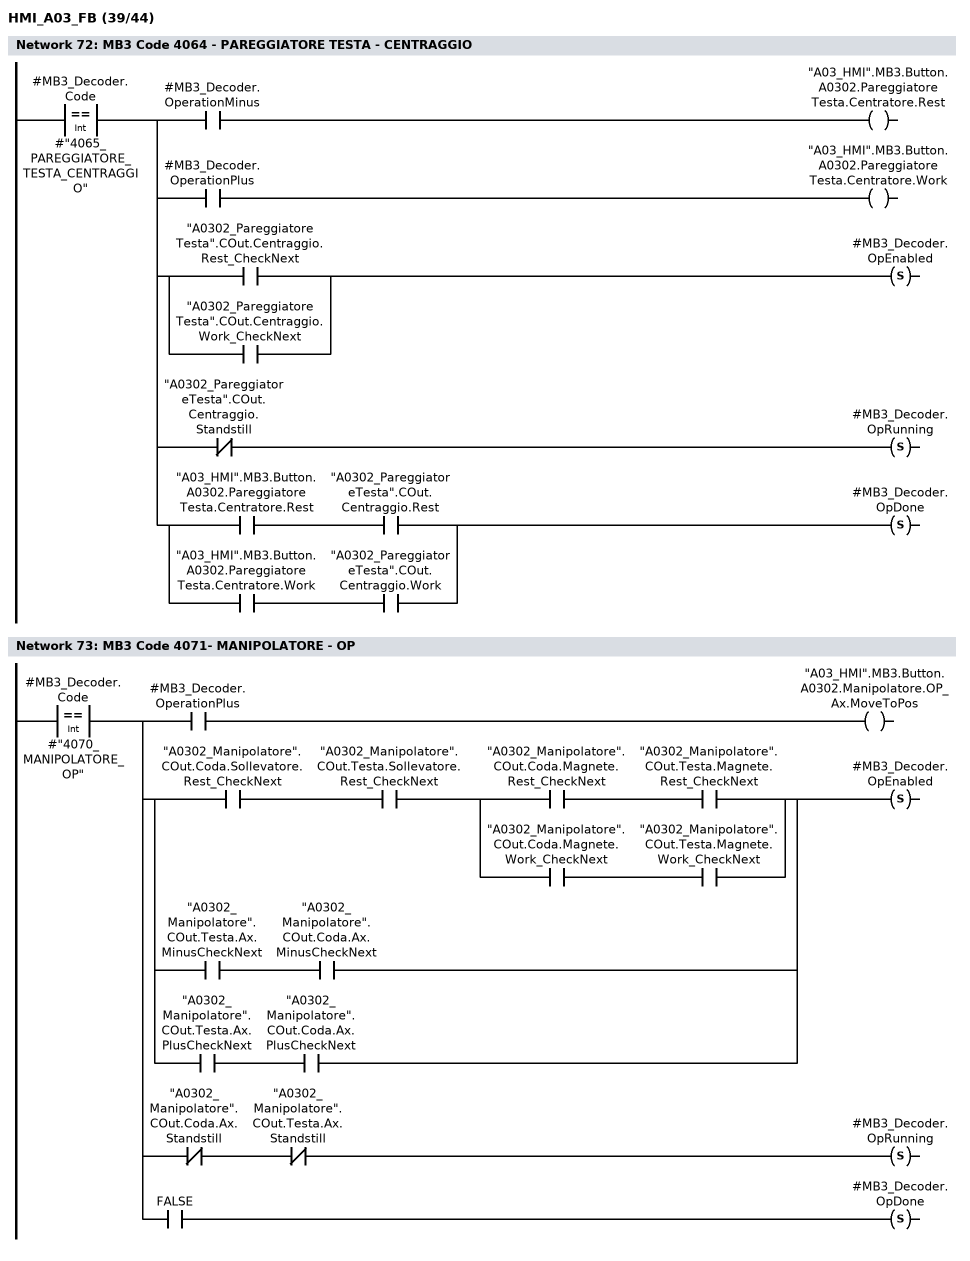
   RUNG wire#powerrail
      { S7_Templates := "SrcType := Int" } EQ_Contact(in1 := #MB3_Decoder.Code, in2 := #"4065_PAREGGIATORE_TESTA_CENTRAGGIO")
      wire#w1
      Contact( #MB3_Decoder.OperationMinus )
      Coil( "A03_HMI".MB3.Button.A0302.PareggiatoreTesta.Centratore.Rest )
   END_RUNG
   RUNG wire#w1
      Contact( #MB3_Decoder.OperationPlus )
      Coil( "A03_HMI".MB3.Button.A0302.PareggiatoreTesta.Centratore.Work )
   END_RUNG
   RUNG wire#w1
      Contact( "A0302_PareggiatoreTesta".COut.Centraggio.Rest_CheckNext )
      wire#w2
      S_Coil( #MB3_Decoder.OpEnabled )
   END_RUNG
   RUNG wire#w1
      Contact( "A0302_PareggiatoreTesta".COut.Centraggio.Work_CheckNext )
   END_RUNG wire#w2
   RUNG wire#w1
      I_Contact( "A0302_PareggiatoreTesta".COut.Centraggio.Standstill )
      S_Coil( #MB3_Decoder.OpRunning )
   END_RUNG
   RUNG wire#w1
      Contact( "A03_HMI".MB3.Button.A0302.PareggiatoreTesta.Centratore.Rest )
      Contact( "A0302_PareggiatoreTesta".COut.Centraggio.Rest )
      wire#w3
      S_Coil( #MB3_Decoder.OpDone )
   END_RUNG
   RUNG wire#w1
      Contact( "A03_HMI".MB3.Button.A0302.PareggiatoreTesta.Centratore.Work )
      Contact( "A0302_PareggiatoreTesta".COut.Centraggio.Work )
   END_RUNG wire#w3
   // the same network as SCL:
   #_w1 := #MB3_Decoder.Code = #"4065_PAREGGIATORE_TESTA_CENTRAGGIO";
   "A03_HMI".MB3.Button.A0302.PareggiatoreTesta.Centratore.Rest := #_w1 AND #MB3_Decoder.OperationMinus;
   "A03_HMI".MB3.Button.A0302.PareggiatoreTesta.Centratore.Work := #_w1 AND #MB3_Decoder.OperationPlus;
   IF #_w1 AND ("A0302_PareggiatoreTesta".COut.Centraggio.Rest_CheckNext OR "A0302_PareggiatoreTesta".COut.Centraggio.Work_CheckNext) THEN
       #MB3_Decoder.OpEnabled := TRUE;
   END_IF;
   IF #_w1 AND NOT "A0302_PareggiatoreTesta".COut.Centraggio.Standstill THEN
       #MB3_Decoder.OpRunning := TRUE;
   END_IF;
   IF #_w1 AND (("A03_HMI".MB3.Button.A0302.PareggiatoreTesta.Centratore.Rest AND "A0302_PareggiatoreTesta".COut.Centraggio.Rest) OR ("A03_HMI".MB3.Button.A0302.PareggiatoreTesta.Centratore.Work AND "A0302_PareggiatoreTesta".COut.Centraggio.Work)) THEN
       #MB3_Decoder.OpDone := TRUE;
   END_IF;
END_REGION

REGION Network 73: MB3 Code 4071- MANIPOLATORE - OP
   RUNG wire#powerrail
      { S7_Templates := "SrcType := Int" } EQ_Contact(in1 := #MB3_Decoder.Code, in2 := #"4070_MANIPOLATORE_OP")
      wire#w1
      Contact( #MB3_Decoder.OperationPlus )
      Coil( "A03_HMI".MB3.Button.A0302.Manipolatore.OP_Ax.MoveToPos )
   END_RUNG
   RUNG wire#w1
      Contact( "A0302_Manipolatore".COut.Coda.Sollevatore.Rest_CheckNext )
      Contact( "A0302_Manipolatore".COut.Testa.Sollevatore.Rest_CheckNext )
      wire#w2
      Contact( "A0302_Manipolatore".COut.Coda.Magnete.Rest_CheckNext )
      Contact( "A0302_Manipolatore".COut.Testa.Magnete.Rest_CheckNext )
      wire#w3
      S_Coil( #MB3_Decoder.OpEnabled )
   END_RUNG
   RUNG wire#w2
      Contact( "A0302_Manipolatore".COut.Coda.Magnete.Work_CheckNext )
      Contact( "A0302_Manipolatore".COut.Testa.Magnete.Work_CheckNext )
   END_RUNG wire#w3
   RUNG wire#w1
      Contact( "A0302_Manipolatore".COut.Testa.Ax.MinusCheckNext )
      Contact( "A0302_Manipolatore".COut.Coda.Ax.MinusCheckNext )
   END_RUNG wire#w3
   RUNG wire#w1
      Contact( "A0302_Manipolatore".COut.Testa.Ax.PlusCheckNext )
      Contact( "A0302_Manipolatore".COut.Coda.Ax.PlusCheckNext )
   END_RUNG wire#w3
   RUNG wire#w1
      I_Contact( "A0302_Manipolatore".COut.Coda.Ax.Standstill )
      I_Contact( "A0302_Manipolatore".COut.Testa.Ax.Standstill )
      S_Coil( #MB3_Decoder.OpRunning )
   END_RUNG
   RUNG wire#w1
      Contact( FALSE )
      S_Coil( #MB3_Decoder.OpDone )
   END_RUNG
   // the same network as SCL:
   #_w1 := #MB3_Decoder.Code = #"4070_MANIPOLATORE_OP";
   "A03_HMI".MB3.Button.A0302.Manipolatore.OP_Ax.MoveToPos := #_w1 AND #MB3_Decoder.OperationPlus;
   IF #_w1 AND (("A0302_Manipolatore".COut.Coda.Sollevatore.Rest_CheckNext AND "A0302_Manipolatore".COut.Testa.Sollevatore.Rest_CheckNext AND (("A0302_Manipolatore".COut.Coda.Magnete.Rest_CheckNext AND "A0302_Manipolatore".COut.Testa.Magnete.Rest_CheckNext) OR ("A0302_Manipolatore".COut.Coda.Magnete.Work_CheckNext AND "A0302_Manipolatore".COut.Testa.Magnete.Work_CheckNext))) OR ("A0302_Manipolatore".COut.Testa.Ax.MinusCheckNext AND "A0302_Manipolatore".COut.Coda.Ax.MinusCheckNext) OR ("A0302_Manipolatore".COut.Testa.Ax.PlusCheckNext AND "A0302_Manipolatore".COut.Coda.Ax.PlusCheckNext)) THEN
       #MB3_Decoder.OpEnabled := TRUE;
   END_IF;
   IF #_w1 AND NOT "A0302_Manipolatore".COut.Coda.Ax.Standstill AND NOT "A0302_Manipolatore".COut.Testa.Ax.Standstill THEN
       #MB3_Decoder.OpRunning := TRUE;
   END_IF;
   IF #_w1 AND FALSE THEN #MB3_Decoder.OpDone := TRUE; END_IF;
END_REGION

REGION Network 74: MB3 Code 4071- MANIPOLATORE -AX
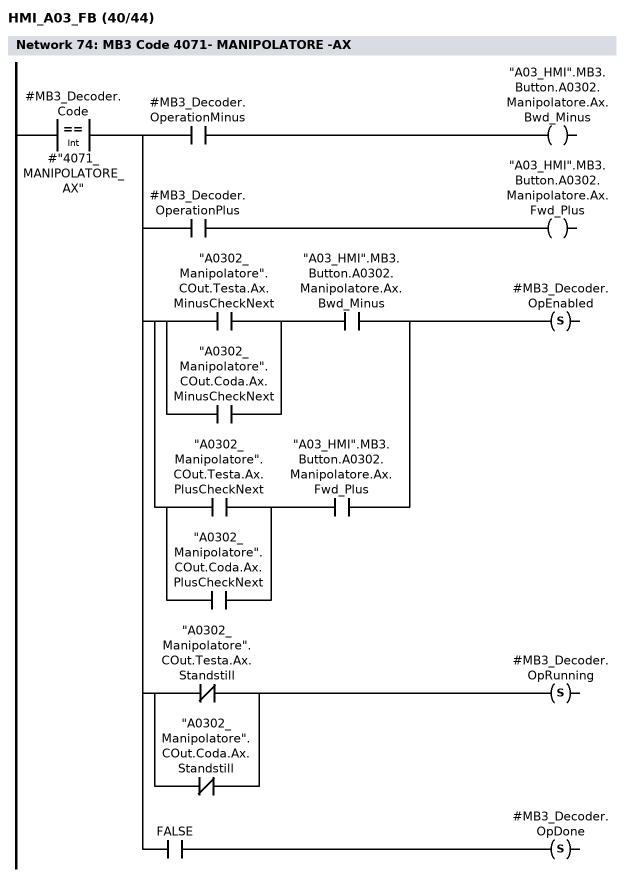
   RUNG wire#powerrail
      { S7_Templates := "SrcType := Int" } EQ_Contact(in1 := #MB3_Decoder.Code, in2 := #"4071_MANIPOLATORE_AX")
      wire#w1
      Contact( #MB3_Decoder.OperationMinus )
      Coil( "A03_HMI".MB3.Button.A0302.Manipolatore.Ax.Bwd_Minus )
   END_RUNG
   RUNG wire#w1
      Contact( #MB3_Decoder.OperationPlus )
      Coil( "A03_HMI".MB3.Button.A0302.Manipolatore.Ax.Fwd_Plus )
   END_RUNG
   RUNG wire#w1
      Contact( "A0302_Manipolatore".COut.Testa.Ax.MinusCheckNext )
      wire#w2
      Contact( "A03_HMI".MB3.Button.A0302.Manipolatore.Ax.Bwd_Minus )
      wire#w3
      S_Coil( #MB3_Decoder.OpEnabled )
   END_RUNG
   RUNG wire#w1
      Contact( "A0302_Manipolatore".COut.Coda.Ax.MinusCheckNext )
   END_RUNG wire#w2
   RUNG wire#w1
      Contact( "A0302_Manipolatore".COut.Testa.Ax.PlusCheckNext )
      wire#w4
      Contact( "A03_HMI".MB3.Button.A0302.Manipolatore.Ax.Fwd_Plus )
   END_RUNG wire#w3
   RUNG wire#w1
      Contact( "A0302_Manipolatore".COut.Coda.Ax.PlusCheckNext )
   END_RUNG wire#w4
   RUNG wire#w1
      I_Contact( "A0302_Manipolatore".COut.Testa.Ax.Standstill )
      wire#w5
      S_Coil( #MB3_Decoder.OpRunning )
   END_RUNG
   RUNG wire#w1
      I_Contact( "A0302_Manipolatore".COut.Coda.Ax.Standstill )
   END_RUNG wire#w5
   RUNG wire#w1
      Contact( FALSE )
      S_Coil( #MB3_Decoder.OpDone )
   END_RUNG
   // the same network as SCL:
   #_w1 := #MB3_Decoder.Code = #"4071_MANIPOLATORE_AX";
   "A03_HMI".MB3.Button.A0302.Manipolatore.Ax.Bwd_Minus := #_w1 AND #MB3_Decoder.OperationMinus;
   "A03_HMI".MB3.Button.A0302.Manipolatore.Ax.Fwd_Plus := #_w1 AND #MB3_Decoder.OperationPlus;
   IF #_w1 AND ((("A0302_Manipolatore".COut.Testa.Ax.MinusCheckNext OR "A0302_Manipolatore".COut.Coda.Ax.MinusCheckNext) AND "A03_HMI".MB3.Button.A0302.Manipolatore.Ax.Bwd_Minus) OR (("A0302_Manipolatore".COut.Testa.Ax.PlusCheckNext OR "A0302_Manipolatore".COut.Coda.Ax.PlusCheckNext) AND "A03_HMI".MB3.Button.A0302.Manipolatore.Ax.Fwd_Plus)) THEN
       #MB3_Decoder.OpEnabled := TRUE;
   END_IF;
   IF #_w1 AND (NOT "A0302_Manipolatore".COut.Testa.Ax.Standstill OR NOT "A0302_Manipolatore".COut.Coda.Ax.Standstill) THEN
       #MB3_Decoder.OpRunning := TRUE;
   END_IF;
   IF #_w1 AND FALSE THEN #MB3_Decoder.OpDone := TRUE; END_IF;
END_REGION

REGION Network 75: MB3 Code 4072- MANIPOLATORE -AX-POS
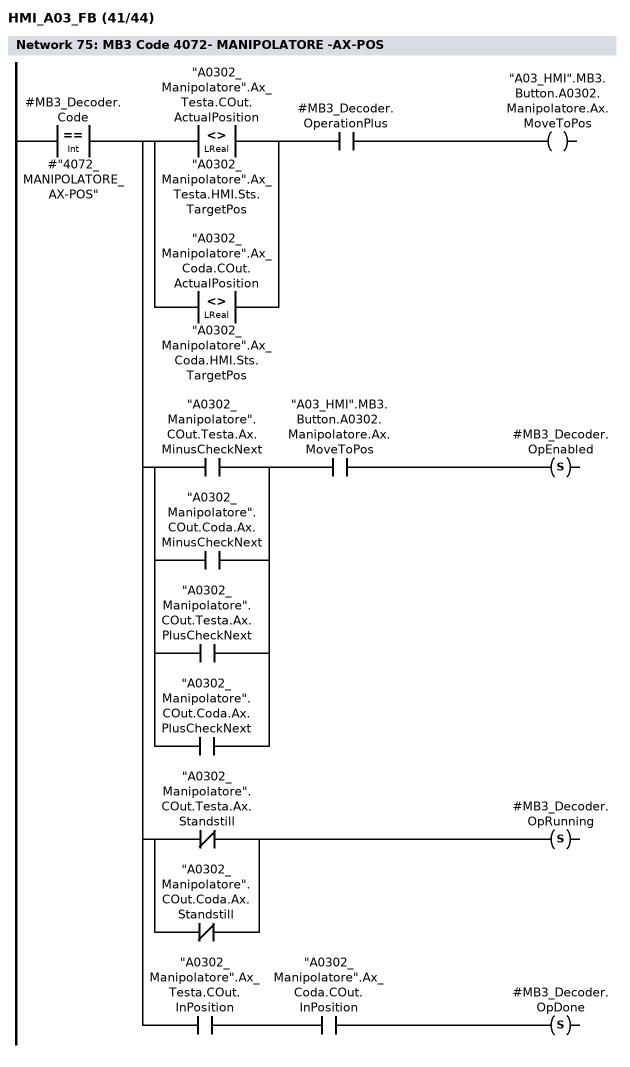
   RUNG wire#powerrail
      { S7_Templates := "SrcType := Int" } EQ_Contact(in1 := #MB3_Decoder.Code, in2 := #"4072_MANIPOLATORE_AX-POS")
      wire#w1
      { S7_Templates := "SrcType := LReal" } NE_Contact(in1 := "A0302_Manipolatore".Ax_Testa.COut.ActualPosition, in2 := "A0302_Manipolatore".Ax_Testa.HMI.Sts.TargetPos)
      wire#w2
      Contact( #MB3_Decoder.OperationPlus )
      Coil( "A03_HMI".MB3.Button.A0302.Manipolatore.Ax.MoveToPos )
   END_RUNG
   RUNG wire#w1
      { S7_Templates := "SrcType := LReal" } NE_Contact(in1 := "A0302_Manipolatore".Ax_Coda.COut.ActualPosition, in2 := "A0302_Manipolatore".Ax_Coda.HMI.Sts.TargetPos)
   END_RUNG wire#w2
   RUNG wire#w1
      Contact( "A0302_Manipolatore".COut.Testa.Ax.MinusCheckNext )
      wire#w3
      Contact( "A03_HMI".MB3.Button.A0302.Manipolatore.Ax.MoveToPos )
      S_Coil( #MB3_Decoder.OpEnabled )
   END_RUNG
   RUNG wire#w1
      Contact( "A0302_Manipolatore".COut.Coda.Ax.MinusCheckNext )
   END_RUNG wire#w3
   RUNG wire#w1
      Contact( "A0302_Manipolatore".COut.Testa.Ax.PlusCheckNext )
   END_RUNG wire#w3
   RUNG wire#w1
      Contact( "A0302_Manipolatore".COut.Coda.Ax.PlusCheckNext )
   END_RUNG wire#w3
   RUNG wire#w1
      I_Contact( "A0302_Manipolatore".COut.Testa.Ax.Standstill )
      wire#w4
      S_Coil( #MB3_Decoder.OpRunning )
   END_RUNG
   RUNG wire#w1
      I_Contact( "A0302_Manipolatore".COut.Coda.Ax.Standstill )
   END_RUNG wire#w4
   RUNG wire#w1
      Contact( "A0302_Manipolatore".Ax_Testa.COut.InPosition )
      Contact( "A0302_Manipolatore".Ax_Coda.COut.InPosition )
      S_Coil( #MB3_Decoder.OpDone )
   END_RUNG
   // the same network as SCL:
   #_w1 := #MB3_Decoder.Code = #"4072_MANIPOLATORE_AX-POS";
   "A03_HMI".MB3.Button.A0302.Manipolatore.Ax.MoveToPos := #_w1 AND (("A0302_Manipolatore".Ax_Testa.COut.ActualPosition <> "A0302_Manipolatore".Ax_Testa.HMI.Sts.TargetPos) OR ("A0302_Manipolatore".Ax_Coda.COut.ActualPosition <> "A0302_Manipolatore".Ax_Coda.HMI.Sts.TargetPos)) AND #MB3_Decoder.OperationPlus;
   IF #_w1 AND ("A0302_Manipolatore".COut.Testa.Ax.MinusCheckNext OR "A0302_Manipolatore".COut.Coda.Ax.MinusCheckNext OR "A0302_Manipolatore".COut.Testa.Ax.PlusCheckNext OR "A0302_Manipolatore".COut.Coda.Ax.PlusCheckNext) AND "A03_HMI".MB3.Button.A0302.Manipolatore.Ax.MoveToPos THEN
       #MB3_Decoder.OpEnabled := TRUE;
   END_IF;
   IF #_w1 AND (NOT "A0302_Manipolatore".COut.Testa.Ax.Standstill OR NOT "A0302_Manipolatore".COut.Coda.Ax.Standstill) THEN
       #MB3_Decoder.OpRunning := TRUE;
   END_IF;
   IF #_w1 AND "A0302_Manipolatore".Ax_Testa.COut.InPosition AND "A0302_Manipolatore".Ax_Coda.COut.InPosition THEN
       #MB3_Decoder.OpDone := TRUE;
   END_IF;
END_REGION

REGION Network 76: MB3 Code 4073 - MANIPOLATORE- MAGNETE
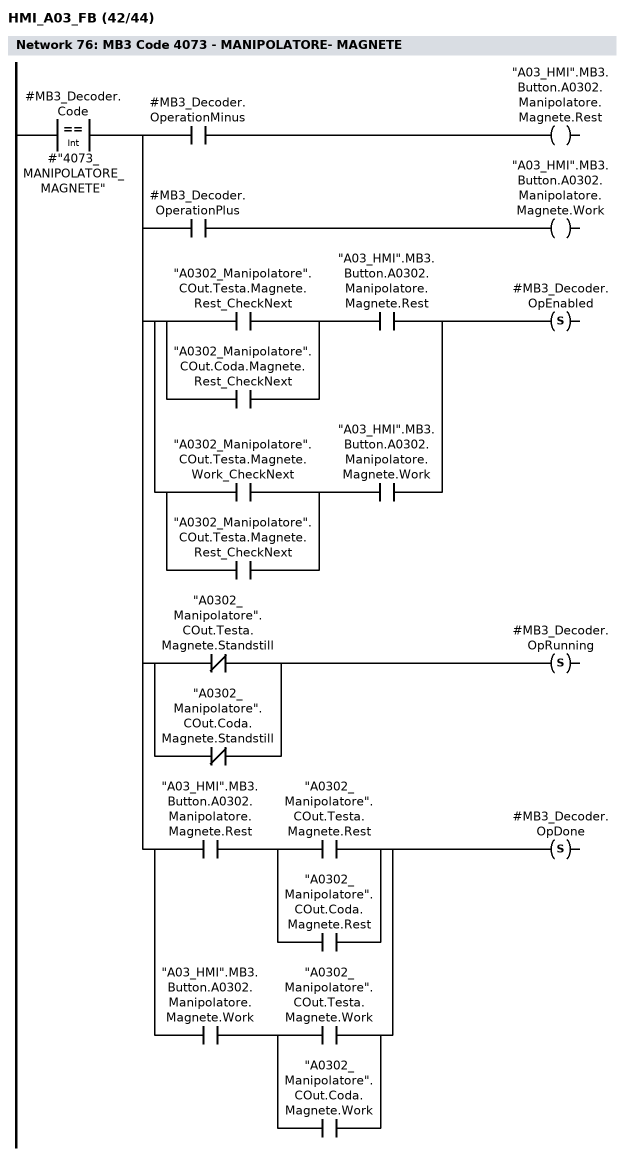
   RUNG wire#powerrail
      { S7_Templates := "SrcType := Int" } EQ_Contact(in1 := #MB3_Decoder.Code, in2 := #"4073_MANIPOLATORE_MAGNETE")
      wire#w1
      Contact( #MB3_Decoder.OperationMinus )
      Coil( "A03_HMI".MB3.Button.A0302.Manipolatore.Magnete.Rest )
   END_RUNG
   RUNG wire#w1
      Contact( #MB3_Decoder.OperationPlus )
      Coil( "A03_HMI".MB3.Button.A0302.Manipolatore.Magnete.Work )
   END_RUNG
   RUNG wire#w1
      Contact( "A0302_Manipolatore".COut.Testa.Magnete.Rest_CheckNext )
      wire#w2
      Contact( "A03_HMI".MB3.Button.A0302.Manipolatore.Magnete.Rest )
      wire#w3
      S_Coil( #MB3_Decoder.OpEnabled )
   END_RUNG
   RUNG wire#w1
      Contact( "A0302_Manipolatore".COut.Coda.Magnete.Rest_CheckNext )
   END_RUNG wire#w2
   RUNG wire#w1
      Contact( "A0302_Manipolatore".COut.Testa.Magnete.Work_CheckNext )
      wire#w4
      Contact( "A03_HMI".MB3.Button.A0302.Manipolatore.Magnete.Work )
   END_RUNG wire#w3
   RUNG wire#w1
      Contact( "A0302_Manipolatore".COut.Testa.Magnete.Rest_CheckNext )
   END_RUNG wire#w4
   RUNG wire#w1
      I_Contact( "A0302_Manipolatore".COut.Testa.Magnete.Standstill )
      wire#w5
      S_Coil( #MB3_Decoder.OpRunning )
   END_RUNG
   RUNG wire#w1
      I_Contact( "A0302_Manipolatore".COut.Coda.Magnete.Standstill )
   END_RUNG wire#w5
   RUNG wire#w1
      Contact( "A03_HMI".MB3.Button.A0302.Manipolatore.Magnete.Rest )
      wire#w6
      Contact( "A0302_Manipolatore".COut.Testa.Magnete.Rest )
      wire#w7
      S_Coil( #MB3_Decoder.OpDone )
   END_RUNG
   RUNG wire#w6
      Contact( "A0302_Manipolatore".COut.Coda.Magnete.Rest )
   END_RUNG wire#w7
   RUNG wire#w1
      Contact( "A03_HMI".MB3.Button.A0302.Manipolatore.Magnete.Work )
      wire#w8
      Contact( "A0302_Manipolatore".COut.Testa.Magnete.Work )
   END_RUNG wire#w7
   RUNG wire#w8
      Contact( "A0302_Manipolatore".COut.Coda.Magnete.Work )
   END_RUNG wire#w7
   // the same network as SCL:
   #_w1 := #MB3_Decoder.Code = #"4073_MANIPOLATORE_MAGNETE";
   "A03_HMI".MB3.Button.A0302.Manipolatore.Magnete.Rest := #_w1 AND #MB3_Decoder.OperationMinus;
   "A03_HMI".MB3.Button.A0302.Manipolatore.Magnete.Work := #_w1 AND #MB3_Decoder.OperationPlus;
   IF #_w1 AND ((("A0302_Manipolatore".COut.Testa.Magnete.Rest_CheckNext OR "A0302_Manipolatore".COut.Coda.Magnete.Rest_CheckNext) AND "A03_HMI".MB3.Button.A0302.Manipolatore.Magnete.Rest) OR (("A0302_Manipolatore".COut.Testa.Magnete.Work_CheckNext OR "A0302_Manipolatore".COut.Testa.Magnete.Rest_CheckNext) AND "A03_HMI".MB3.Button.A0302.Manipolatore.Magnete.Work)) THEN
       #MB3_Decoder.OpEnabled := TRUE;
   END_IF;
   IF #_w1 AND (NOT "A0302_Manipolatore".COut.Testa.Magnete.Standstill OR NOT "A0302_Manipolatore".COut.Coda.Magnete.Standstill) THEN
       #MB3_Decoder.OpRunning := TRUE;
   END_IF;
   IF #_w1 AND (("A03_HMI".MB3.Button.A0302.Manipolatore.Magnete.Rest AND ("A0302_Manipolatore".COut.Testa.Magnete.Rest OR "A0302_Manipolatore".COut.Coda.Magnete.Rest)) OR ("A03_HMI".MB3.Button.A0302.Manipolatore.Magnete.Work AND ("A0302_Manipolatore".COut.Testa.Magnete.Work OR "A0302_Manipolatore".COut.Coda.Magnete.Work))) THEN
       #MB3_Decoder.OpDone := TRUE;
   END_IF;
END_REGION

REGION Network 77: MB3 Code 4074 - MANIPOLATORE- SOLLEVATORE
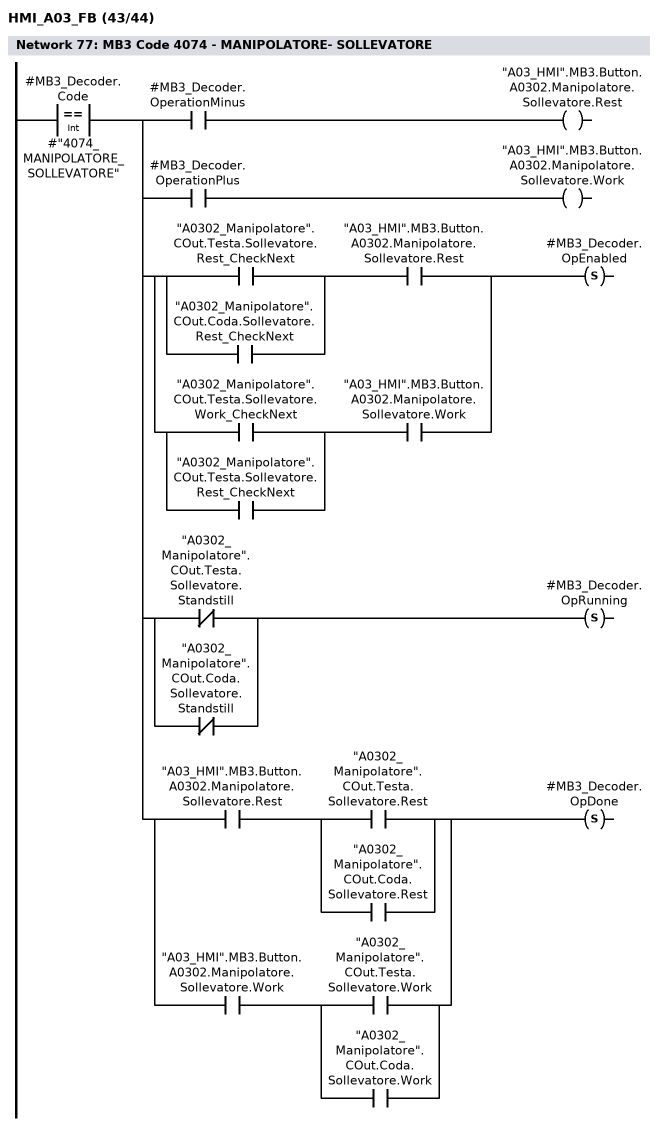
   RUNG wire#powerrail
      { S7_Templates := "SrcType := Int" } EQ_Contact(in1 := #MB3_Decoder.Code, in2 := #"4074_MANIPOLATORE_SOLLEVATORE")
      wire#w1
      Contact( #MB3_Decoder.OperationMinus )
      Coil( "A03_HMI".MB3.Button.A0302.Manipolatore.Sollevatore.Rest )
   END_RUNG
   RUNG wire#w1
      Contact( #MB3_Decoder.OperationPlus )
      Coil( "A03_HMI".MB3.Button.A0302.Manipolatore.Sollevatore.Work )
   END_RUNG
   RUNG wire#w1
      Contact( "A0302_Manipolatore".COut.Testa.Sollevatore.Rest_CheckNext )
      wire#w2
      Contact( "A03_HMI".MB3.Button.A0302.Manipolatore.Sollevatore.Rest )
      wire#w3
      S_Coil( #MB3_Decoder.OpEnabled )
   END_RUNG
   RUNG wire#w1
      Contact( "A0302_Manipolatore".COut.Coda.Sollevatore.Rest_CheckNext )
   END_RUNG wire#w2
   RUNG wire#w1
      Contact( "A0302_Manipolatore".COut.Testa.Sollevatore.Work_CheckNext )
      wire#w4
      Contact( "A03_HMI".MB3.Button.A0302.Manipolatore.Sollevatore.Work )
   END_RUNG wire#w3
   RUNG wire#w1
      Contact( "A0302_Manipolatore".COut.Testa.Sollevatore.Rest_CheckNext )
   END_RUNG wire#w4
   RUNG wire#w1
      I_Contact( "A0302_Manipolatore".COut.Testa.Sollevatore.Standstill )
      wire#w5
      S_Coil( #MB3_Decoder.OpRunning )
   END_RUNG
   RUNG wire#w1
      I_Contact( "A0302_Manipolatore".COut.Coda.Sollevatore.Standstill )
   END_RUNG wire#w5
   RUNG wire#w1
      Contact( "A03_HMI".MB3.Button.A0302.Manipolatore.Sollevatore.Rest )
      wire#w6
      Contact( "A0302_Manipolatore".COut.Testa.Sollevatore.Rest )
      wire#w7
      S_Coil( #MB3_Decoder.OpDone )
   END_RUNG
   RUNG wire#w6
      Contact( "A0302_Manipolatore".COut.Coda.Sollevatore.Rest )
   END_RUNG wire#w7
   RUNG wire#w1
      Contact( "A03_HMI".MB3.Button.A0302.Manipolatore.Sollevatore.Work )
      wire#w8
      Contact( "A0302_Manipolatore".COut.Testa.Sollevatore.Work )
   END_RUNG wire#w7
   RUNG wire#w8
      Contact( "A0302_Manipolatore".COut.Coda.Sollevatore.Work )
   END_RUNG wire#w7
   // the same network as SCL:
   #_w1 := #MB3_Decoder.Code = #"4074_MANIPOLATORE_SOLLEVATORE";
   "A03_HMI".MB3.Button.A0302.Manipolatore.Sollevatore.Rest := #_w1 AND #MB3_Decoder.OperationMinus;
   "A03_HMI".MB3.Button.A0302.Manipolatore.Sollevatore.Work := #_w1 AND #MB3_Decoder.OperationPlus;
   IF #_w1 AND ((("A0302_Manipolatore".COut.Testa.Sollevatore.Rest_CheckNext OR "A0302_Manipolatore".COut.Coda.Sollevatore.Rest_CheckNext) AND "A03_HMI".MB3.Button.A0302.Manipolatore.Sollevatore.Rest) OR (("A0302_Manipolatore".COut.Testa.Sollevatore.Work_CheckNext OR "A0302_Manipolatore".COut.Testa.Sollevatore.Rest_CheckNext) AND "A03_HMI".MB3.Button.A0302.Manipolatore.Sollevatore.Work)) THEN
       #MB3_Decoder.OpEnabled := TRUE;
   END_IF;
   IF #_w1 AND (NOT "A0302_Manipolatore".COut.Testa.Sollevatore.Standstill OR NOT "A0302_Manipolatore".COut.Coda.Sollevatore.Standstill) THEN
       #MB3_Decoder.OpRunning := TRUE;
   END_IF;
   IF #_w1 AND (("A03_HMI".MB3.Button.A0302.Manipolatore.Sollevatore.Rest AND ("A0302_Manipolatore".COut.Testa.Sollevatore.Rest OR "A0302_Manipolatore".COut.Coda.Sollevatore.Rest)) OR ("A03_HMI".MB3.Button.A0302.Manipolatore.Sollevatore.Work AND ("A0302_Manipolatore".COut.Testa.Sollevatore.Work OR "A0302_Manipolatore".COut.Coda.Sollevatore.Work))) THEN
       #MB3_Decoder.OpDone := TRUE;
   END_IF;
END_REGION

REGION Network 79: >
END_REGION

REGION Network 80: >
END_REGION

REGION Network 81: >
END_REGION

REGION Network 82: MB3 Decoder
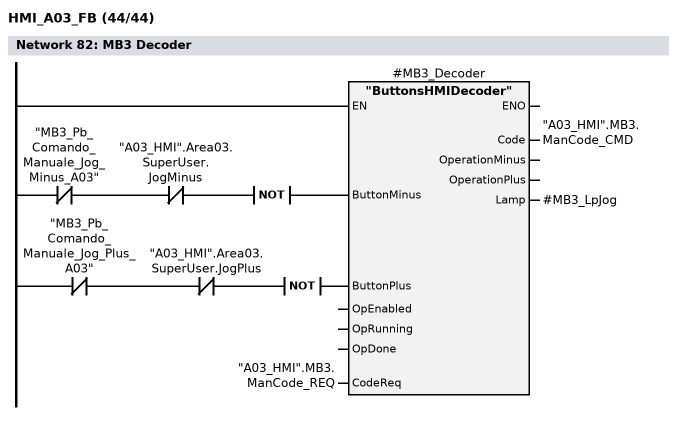
   RUNG wire#powerrail
      #MB3_Decoder(ButtonMinus := wire#w1, ButtonPlus := wire#w2, OpEnabled :=, OpRunning :=, OpDone :=, CodeReq := "A03_HMI".MB3.ManCode_REQ, Code => "A03_HMI".MB3.ManCode_CMD, OperationMinus =>, OperationPlus =>, Lamp => #MB3_LpJog)
   END_RUNG
   RUNG wire#powerrail
      I_Contact( "MB3_Pb_Comando_Manuale_Jog_Minus_A03" )
      I_Contact( "A03_HMI".Area03.SuperUser.JogMinus )
      Not()
   END_RUNG wire#w1
   RUNG wire#powerrail
      I_Contact( "MB3_Pb_Comando_Manuale_Jog_Plus_A03" )
      I_Contact( "A03_HMI".Area03.SuperUser.JogPlus )
      Not()
   END_RUNG wire#w2
   // the same network as SCL:
   #MB3_Decoder(ButtonMinus := NOT (NOT "MB3_Pb_Comando_Manuale_Jog_Minus_A03" AND NOT "A03_HMI".Area03.SuperUser.JogMinus),   // "ButtonsHMIDecoder"
                ButtonPlus := NOT (NOT "MB3_Pb_Comando_Manuale_Jog_Plus_A03" AND NOT "A03_HMI".Area03.SuperUser.JogPlus),
                CodeReq := "A03_HMI".MB3.ManCode_REQ,
                Code => "A03_HMI".MB3.ManCode_CMD,
                Lamp => #MB3_LpJog);
END_REGION
END_FUNCTION_BLOCK

FUNCTION "A03_TrkManager_CALL" : Void   // FC87, LAD
// stored: SetENOAutomatically false
BEGIN

REGION Network 1
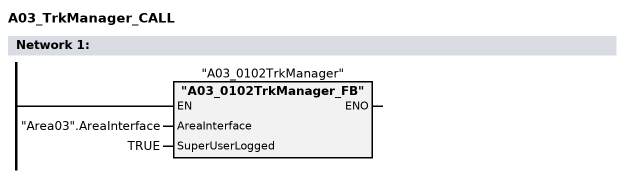
   RUNG wire#powerrail
      "A03_0102TrkManager"(AreaInterface := "Area03".AreaInterface, SuperUserLogged := TRUE)
   END_RUNG
   // the same network as SCL:
   "A03_0102TrkManager"(AreaInterface := "Area03".AreaInterface, SuperUserLogged := TRUE);   // "A03_0102TrkManager_FB"
END_REGION
END_FUNCTION

FUNCTION "A0301_SelSensorON" : Bool   // FC135, LAD
// stored: SetENOAutomatically false
   VAR_INPUT
      SensorsToUse : Array[1..3] of Bool;   // Configurazione sensori selezionati per la lettura del pezzo
      S_Ing : Array[1..3] of Bool;   // IO - Sensori di ingresso Pin di arrivo
   END_VAR
   VAR_TEMP
      "Case" : Int;
      Sens_OK : Bool;
      StsSensPinOK : Array[1..3] of Bool;
   END_VAR
BEGIN

REGION Network 1 (SCL)
   // == CONTROLLO I/O SENSORI INGRESSO FERMI IN BASE ALLA CONFIGURAZIONE ===
   // 

   IF #SensorsToUse[1] AND #S_Ing[1] THEN
       #StsSensPinOK[1] := 1;
   ELSIF (NOT #SensorsToUse[1] OR NOT #S_Ing[1]) THEN
       #StsSensPinOK[1] := 0;
   END_IF;


   IF #SensorsToUse[2] AND #S_Ing[2] THEN
       #StsSensPinOK[2] := 1;
   ELSIF (NOT #SensorsToUse[2] OR NOT #S_Ing[2]) THEN
       #StsSensPinOK[2] := 0;
   END_IF;


   IF #SensorsToUse[3] AND #S_Ing[3] THEN
       #StsSensPinOK[3] := 1;
   ELSIF (NOT #SensorsToUse[3] OR NOT #S_Ing[3]) THEN
       #StsSensPinOK[3] := 0;
   END_IF;
END_REGION

REGION Network 2 (SCL)
   // CONTROLLO ABILITAZIONE SENSORI E STATO SENSORI PER DETERMINARE SE IL CONTROLLO è ANDATO A BUON FINE


    // Controllo con 0 sensori abilitati reset stato sensori
           IF NOT #SensorsToUse[1] AND NOT #SensorsToUse[2] AND NOT #SensorsToUse[3] THEN
               #Sens_OK := 0;

           END_IF;

           // Controllo con 1 sensore abilitato   

           IF #SensorsToUse[1] AND NOT #SensorsToUse[2] AND NOT #SensorsToUse[3]
               AND #StsSensPinOK[1] THEN
               #Sens_OK := 1;

           END_IF;

   // Controllo con 2 sensori abilitati
           IF #SensorsToUse[1] AND #SensorsToUse[2] AND NOT #SensorsToUse[3]
               AND #StsSensPinOK[1] AND #StsSensPinOK[2] THEN
               #Sens_OK := 1;

           END_IF;

    // Controllo con 3 sensori abilitati
           IF #SensorsToUse[1] AND #SensorsToUse[2] AND #SensorsToUse[3]
               AND #StsSensPinOK[1] AND #StsSensPinOK[2] AND #StsSensPinOK[3] THEN
               #Sens_OK := 1;

           END_IF;

    // Controllo con 2 sensori abilitati non in appoggio
           IF NOT #SensorsToUse[1] AND #SensorsToUse[2] AND #SensorsToUse[3]
               AND NOT #StsSensPinOK[1] AND #StsSensPinOK[2] AND #StsSensPinOK[3] THEN
               #Sens_OK := 1;

           END_IF;
END_REGION

REGION Network 3
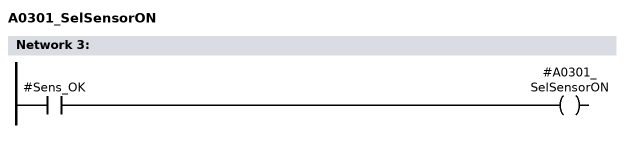
   RUNG wire#powerrail
      Contact( #Sens_OK )
      Coil( #A0301_SelSensorON )
   END_RUNG
   // the same network as SCL:
   #A0301_SelSensorON := #Sens_OK;
END_REGION
END_FUNCTION

FUNCTION "A0301_Manager_CALL" : Void   // FC59, LAD
// stored: SetENOAutomatically false
BEGIN

REGION Network 2 (SCL): << TRASFERIMENTO stati CIn del blocco >>
   // TRASFERIMENTO CIn TRASPORTO
   "A0301_Manager".CIn.Trasporto := "A0301_Trasporto".COut.Ax;

   // TRASFERIMENTO Cin UTENZE FERMI P1
   "A0301_Manager".CIn.P1.Fermi := "A0301_Fermi_P1".COut.Fermi;
   "A0301_Manager".CIn.P1.Sfalsatore := "A0301_Fermi_P1".COut.Pareggiatore;

   // TRASFERIMENTO CIn UTENZE FERMI P2
   "A0301_Manager".CIn.P2.Fermi := "A0301_Fermi_P2".COut.Fermi;
   "A0301_Manager".CIn.P2.Sollevatore := "A0301_Fermi_P2".COut.Sollevatori;

   // TRASFERIMENTO CIn UTENZE FERMI P3
   "A0301_Manager".CIn.P3.Fermi := "A0301_Fermi_P3".COut.Fermi;

   // TRASFERIMENTO CIn UTENZE RIBALTATORE
   "A0301_Manager".CIn.Ribaltatore.Solleva_Rib := "A0301_Ribaltatore".COut.Solleva_Rib;
   "A0301_Manager".CIn.Ribaltatore.Ax := "A0301_Ribaltatore".COut.Ribaltatore;
   "A0301_Manager".CIn.Ribaltatore.Sts_Ribaltatore := "A0301_Ribaltatore".COut.Ribaltatore_Sts;

   // TRASFERIMENTO CIn UTENZE FERMI P4
   "A0301_Manager".CIn.P4.Fermi := "A0301_Fermi_P4".COut.Fermi;

   // TRASFERIMENTO CIn UTENZE FERMI P5
   "A0301_Manager".CIn.P5.Spintore_Lat.Spin_Lat1 := "A0301_Spintore_Lat".COut.Spin_Lat1;
   "A0301_Manager".CIn.P5.Spintore_Lat.Spin_Lat2 := "A0301_Spintore_Lat".COut.Spin_Lat2;
   "A0301_Manager".CIn.P5.Spintore_Lat.Vrt_1 := "A0301_Spintore_Lat".COut.Vrt_1;
   "A0301_Manager".CIn.P5.Spintore_Lat.Orz_1 := "A0301_Spintore_Lat".COut.Orz_1;
   "A0301_Manager".CIn.P5.Spintore_Lat.Vrt_2 := "A0301_Spintore_Lat".COut.Vrt_2;
   "A0301_Manager".CIn.P5.Spintore_Lat.Orz_2 := "A0301_Spintore_Lat".COut.Orz_2;
   "A0301_Manager".CIn.P5.Sollevatori := "A0301_Spintore_Lat".COut.Sollevatori;
   "A0301_Manager".CIn.P5.SensUscitaBanco := "A0302_Spintore".IEC.FTC_On;

   // TRASFERIMENTO CIn UTENZE SPINTORE LONGITUDINALE

   "A0301_Manager".CIn.SpintoreLong.Spin_Ev := "A0302_Spintore".COut.Spintore;

   "A0301_Manager".CIn.SpintoreLong.Ax_Sts.PosAttesa_Reached := "A0302_Spintore".COut.Ax_Sts.PosAttesa_Reached;
   "A0301_Manager".CIn.SpintoreLong.Ax_Sts.PosFineSpinta_Reached := "A0302_Spintore".COut.Ax_Sts.PosFineSpinta_Reached;

   // Production Mng
   "A0301_Manager".CIn.ProdManager := "Areas_ITF".Prod.A03_A04;
END_REGION

REGION Network 3 (SCL): << TRASFERIMENTO stati DataIn del blocco >>
   // SOSTITUIRE Sys.ByPass  CON INGRESSI DIGITALI
   //
   // MB3 Pulsante semiautomatico 
   "A0301_Manager".DataIn.SemiAut_Pb := "MB3_Pb_Avanti_Stazione_1_Area03";

   REGION TRASFERIMENTO DataIn SENSORI INGRESSO USCITA P1
       // PRESENZA PEZZO INGRESSO
       "A0301_Manager".DataIn.P1.Sens_Ing[1] := "A0301_Cinghia_1_Phc_1";
       "A0301_Manager".DataIn.P1.Sens_Ing[2] := "A0301_Cinghia_2_Phc_1";
       "A0301_Manager".DataIn.P1.Sens_Ing[3] := "A0301_Cinghia_4_Phc_1";
       // USCITA PEZZO
       "A0301_Manager".DataIn.P1.Sens_Out[1] := "A0301_Cinghia_1_Phc_2";
       "A0301_Manager".DataIn.P1.Sens_Out[2] := "A0301_Cinghia_2_Phc_2";
       "A0301_Manager".DataIn.P1.Sens_Out[3] := "A0301_Cinghia_4_Phc_2";
   END_REGION ;

   REGION TRASFERIMENTO DataIn SENSORI INGRESSO USCITA P2
       // PRESENZA PEZZO INGRESSO
       "A0301_Manager".DataIn.P2.Sens_Ing[1] := "A0301_Cinghia_1_Phc_3";
       "A0301_Manager".DataIn.P2.Sens_Ing[2] := "A0301_Cinghia_2_Phc_3";
       "A0301_Manager".DataIn.P2.Sens_Ing[3] := "A0301_Cinghia_4_Phc_3";
       // USCITA PEZZO solo PREDISPOSTO
       "A0301_Manager".DataIn.P2.Sens_Out[1] := "Sys".ByPass;
       "A0301_Manager".DataIn.P2.Sens_Out[2] := "Sys".ByPass;
       "A0301_Manager".DataIn.P2.Sens_Out[3] := "Sys".ByPass;
   END_REGION ;

   REGION TRASFERIMENTO DataIn SENSORI INGRESSO USCITA P3
       // PRESENZA PEZZO INGRESSO
       "A0301_Manager".DataIn.P3.Sens_Ing[1] := "A0301_Cinghia_1_Phc_5";
       "A0301_Manager".DataIn.P3.Sens_Ing[2] := "A0301_Cinghia_2_Phc_5";
       "A0301_Manager".DataIn.P3.Sens_Ing[3] := "A0301_Cinghia_4_Phc_5";
       // USCITA PEZZO
       "A0301_Manager".DataIn.P3.Sens_Out[1] := "A0301_Cinghia_1_Phc_6";
       "A0301_Manager".DataIn.P3.Sens_Out[2] := "A0301_Cinghia_2_Phc_6";
       "A0301_Manager".DataIn.P3.Sens_Out[3] := "A0301_Cinghia_4_Phc_6";
   END_REGION ;

   REGION TRASFERIMENTO DataIn SENSORI INGRESSO USCITA P4
       // PRESENZA PEZZO INGRESSO
       "A0301_Manager".DataIn.P4.Sens_Ing[1] := "A0301_Cinghia_1_Phc_7";
       "A0301_Manager".DataIn.P4.Sens_Ing[2] := "A0301_Cinghia_2_Phc_7";
       "A0301_Manager".DataIn.P4.Sens_Ing[3] := "A0301_Cinghia_4_Phc_7";
       // USCITA PEZZO
       "A0301_Manager".DataIn.P4.Sens_Out[1] := "A0301_Cinghia_1_Phc_8";
       "A0301_Manager".DataIn.P4.Sens_Out[2] := "A0301_Cinghia_2_Phc_8";
       "A0301_Manager".DataIn.P4.Sens_Out[3] := "A0301_Cinghia_4_Phc_8";
   END_REGION ;

   //  TRASFERIMENTO DataIn SENSORI USCITA BANCO P5
   "A0301_Manager".DataIn.P5.Sens_Fuori_Ingombro_A0301 := "A0302_Spintore".IEC.FTC_On;
END_REGION

REGION Network 4: << Machine Call >>
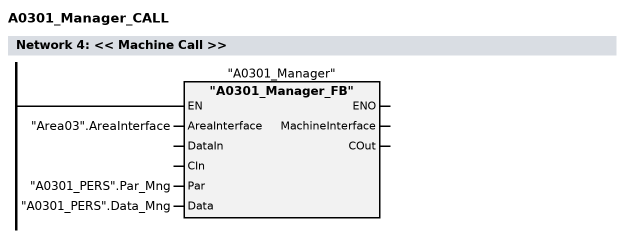
   RUNG wire#powerrail
      "A0301_Manager"(AreaInterface := "Area03".AreaInterface, DataIn :=, CIn :=, Par := "A0301_PERS".Par_Mng, Data := "A0301_PERS".Data_Mng, MachineInterface =>, COut =>)
   END_RUNG
   // the same network as SCL:
   "A0301_Manager"(AreaInterface := "Area03".AreaInterface,   // "A0301_Manager_FB"
                   Par := "A0301_PERS".Par_Mng,
                   Data := "A0301_PERS".Data_Mng);
END_REGION
END_FUNCTION

FUNCTION_BLOCK "A0301_Manager_FB"   // FB45, LAD
TITLE = == A03 STATION RECIVE PRODUCT ==
// stored: MemoryReserve 100, SetENOAutomatically false
   VAR_INPUT
      AreaInterface : "AreaInterface";
      DataIn : Struct
         SemiAut_Pb : Bool;
         P1 : Struct
            Sens_Ing : Array[1..3] of Bool;
            Sens_Out : Array[1..3] of Bool;
         END_STRUCT;
         P2 : Struct
            Sens_Ing : Array[1..3] of Bool;
            Sens_Out : Array[1..3] of Bool;
         END_STRUCT;
         P3 : Struct
            Sens_Ing : Array[1..3] of Bool;
            Sens_Out : Array[1..3] of Bool;
         END_STRUCT;
         P4 : Struct
            Sens_Ing : Array[1..3] of Bool;
            Sens_Out : Array[1..3] of Bool;
         END_STRUCT;
         P5 : Struct
            Sens_Fuori_Ingombro_A0301 : Bool;
         END_STRUCT;
      END_STRUCT;
      CIn : Struct
         Trasporto : "SpeedMachine_COut";
         P1 : Struct
            Fermi : "ValveMachine_COut";
            Sfalsatore : "ValveMachine_COut";
         END_STRUCT;
         P2 : Struct
            Fermi : "ValveMachine_COut";
            Sollevatore : "ValveMachine_COut";
         END_STRUCT;
         P3 : Struct
            Fermi : "ValveMachine_COut";
         END_STRUCT;
         P4 : Struct
            Fermi : "ValveMachine_COut";
         END_STRUCT;
         P5 : Struct
            Sollevatori { ExternalAccessible := 'False'; ExternalVisible := 'False'; ExternalWritable := 'False'} : "ValveMachine_COut";
            Spintore_Lat : Struct
               Spin_Lat1 : Struct
                  Standstill : Bool;
                  Rest_CheckNext : Bool;
                  Work_CheckNext : Bool;
                  Rest : Bool;
                  Work : Bool;
               END_STRUCT;
               Spin_Lat2 : Struct
                  Standstill : Bool;
                  Rest_CheckNext : Bool;
                  Work_CheckNext : Bool;
                  Rest : Bool;
                  Work : Bool;
               END_STRUCT;
               Vrt_1 : "ValveMachine_COut";
               Orz_1 : "ValveMachine_COut";
               Vrt_2 : "ValveMachine_COut";
               Orz_2 : "ValveMachine_COut";
            END_STRUCT;
            SpintoreLong { ExternalAccessible := 'False'; ExternalVisible := 'False'; ExternalWritable := 'False'} : Struct   // Spintore Longitudinale
               Ax : "Positioning_EPOS_Machine_COut";
               Vert : "ValveMachine_COut";
            END_STRUCT;
            SensUscitaBanco : Bool;
         END_STRUCT;
         Ribaltatore : Struct
            Solleva_Rib : "ValveMachine_COut";
            Ax : "Positioning_EPOS_Machine_COut";
            Sts_Ribaltatore : Struct
               Pos0_Reached : Bool;
               Pos1_Reached : Bool;
               Pos2_Reached : Bool;
               Pos3_Reached : Bool;
            END_STRUCT;
         END_STRUCT;
         SpintoreLong : Struct
            Ax_Sts { ExternalAccessible := 'False'; ExternalVisible := 'False'; ExternalWritable := 'False'} : Struct
               PosAttesa_Reached : Bool;
               PosFineSpinta_Reached : Bool;
            END_STRUCT;
            Spin_Ev : "ValveMachine_COut";
         END_STRUCT;
         ProdManager : "Prod_Beam_Ctrl";
      END_STRUCT;
   END_VAR
   VAR_OUTPUT
      MachineInterface : "MachineInterface";
      COut : Struct
         P1 : Struct
            Fermi : "ValveMachine_Manager";
            Pareggiatore : "ValveMachine_Manager";
            ReqPTrk_A02 : Bool;   // Richiesta pezzo ad Area 02
         END_STRUCT;
         P2 : Struct
            Fermi : "ValveMachine_Manager";
            Sollevatore : "ValveMachine_Manager";
         END_STRUCT;
         P3 : Struct
            Fermi : "ValveMachine_Manager";
         END_STRUCT;
         P4 : Struct
            Fermi : "ValveMachine_Manager";
         END_STRUCT;
         P5 : Struct
            Spintore_Lat_1 { ExternalAccessible := 'False'; ExternalVisible := 'False'; ExternalWritable := 'False'} : "ValveMachine_Manager";
            Spintore_Lat_2 { ExternalAccessible := 'False'; ExternalVisible := 'False'; ExternalWritable := 'False'} : "ValveMachine_Manager";
            Sollevatori : "ValveMachine_Manager";
         END_STRUCT;
         Trasporto : "SpeedMachine_CIn_Manager";
         Trasporto_Brw_Req : Bool;
         Trasporto_Frw_Req : Bool;
         Ribaltatore : Struct
            Solleva : "ValveMachine_Manager";
            Ax : "Positioning_EPOS_Machine_Manager";
            Ax_Req : Struct
               Pos0 : Bool;
               Pos1 : Bool;
               Pos2 : Bool;
               Pos3 : Bool;
            END_STRUCT;
            Solleva_REST_Req : Bool;
            Solleva_WORK_Req : Bool;
         END_STRUCT;
      END_STRUCT;
   END_VAR
   VAR_IN_OUT
      Par : Struct
         DlySensorsON : Time;   // [ms] Ritrado ON sensori prima e dopo fermi
         DlySensorsOFF : Time;   // [ms] Ritrado OFF sensori prima e dopo fermi
         TRK : Struct
            BTrk_MoveP4Exit : Time;
            BTrk_MoveToP5 : Time;
         END_STRUCT;
      END_STRUCT;
      Data : Struct
         LastCounter_PartMove_P2toP4 : LReal;
         LastCounter_PartMove_P1toP2 : LReal;
         LastCounter_PartMove_P1toP3 : LReal;
      END_STRUCT;
   END_VAR
   VAR
      Alarm : Struct
         WrongShiftDone { S7_SetPoint := 'True'} : Bool;
         P2toP4_NotReached : Bool;
         P1toP2_NotReached : Bool;
         P1toP3_NotReached : Bool;
         PTrk_TO_BTrk : Struct
            Status : USInt;
         END_STRUCT;
         STOP_FineTurno : Bool;
         STOP_End_Of_Proroduction : Bool;
         STOP_ControlloQualita : Bool;
      END_STRUCT;
      Sts : Struct
         SemiAut : Struct
            ON : Bool;
            Request : Bool;
            MaterialFrw : Bool;
         END_STRUCT;
         P1 : Struct
            Fermi : Struct
               Sens_Ing : Bool;   // 1= Sensori attivati in base alla selezione attiva in base alla lunghezza del pezzo
               Sens_Out : Bool;   // 1= Sensori attivati in base alla selezione attiva in base alla lunghezza del pezzo
            END_STRUCT;
            Sfalsatura_OK : Bool;
         END_STRUCT;
         P2 : Struct
            Fermi : Struct
               Some_Sens_Ing : Bool;   // 1= Alcuni sensori in ingresso alla stanzione sono attivi, ma non tutti
               Sens_Ing : Bool;   // 1= Sensori attivati in base alla selezione attiva in base alla lunghezza del pezzo
               Sens_Out : Bool;   // 1= Sensori attivati in base alla selezione attiva in base alla lunghezza del pezzo
            END_STRUCT;
         END_STRUCT;
         P3 : Struct
            Fermi : Struct
               Some_Sens_Ing : Bool;   // 1= Alcuni sensori in ingresso alla stanzione sono attivi, ma non tutti
               Sens_Ing : Bool;   // 1= Sensori attivati in base alla selezione attiva in base alla lunghezza del pezzo
               Sens_Out : Bool;   // 1= Sensori attivati in base alla selezione attiva in base alla lunghezza del pezzo
            END_STRUCT;
         END_STRUCT;
         P4 : Struct
            Fermi : Struct
               Some_Sens_Ing : Bool;   // 1= Alcuni sensori in ingresso alla stanzione sono attivi, ma non tutti
               Sens_Ing : Bool;   // 1= Sensori attivati in base alla selezione attiva in base alla lunghezza del pezzo
               Sens_Out : Bool;   // 1= Sensori attivati in base alla selezione attiva in base alla lunghezza del pezzo
            END_STRUCT;
         END_STRUCT;
         A0301_Station1 : Struct
            ZoneEmpty { ExternalAccessible := 'False'; ExternalVisible := 'False'; ExternalWritable := 'False'} : Bool;
            Trk { ExternalAccessible := 'False'; ExternalVisible := 'False'; ExternalWritable := 'False'} : Struct
               Actual_O_ID : DInt;
               OLD_OID : DInt;
               A0301_PTrk_Absence : Bool;
               A0301_BTrk_Absence : Bool;
               Wait_A0301_Recive : Bool;   // Attesa ricevimento nuovo O_ID in ingresso su Pos.1 fino a che la Stazione non è vuota dal OLD_ID
            END_STRUCT;
         END_STRUCT;
         Attrezzamento : Struct
            Ready : Bool;
            FindNewID : Bool;
            RequestNewPosition : Bool;
            OLD_OID : DInt;
         END_STRUCT;
         AlarmsPresence : Bool;
         WarningsPresence : Bool;
         IsStandstill : Bool;
      END_STRUCT;
      Ctrl : Struct
         Stop : Bool;
         TRK : Struct
            PTrk : Struct
               Start_Brw : Bool;
               Start_Frw : Bool;
               Pos1_TO_Pos3 : Bool;
               Pos1_TO_Pos2 : Bool;
               Pos2Entry_TO_Pos2Solleva : Bool;
               Paregg_Pos1_to_Pos2 : Bool;
               Paregg_Pos1_to_Pos3 : Bool;
            END_STRUCT;
            BTrk : Struct
               Pos2Up_TO_Pos2Down : Bool;
               WritePos2Up_TO_Pos2Down : Bool;
               Pos4_Entry_TO_Pos4_Exit : Bool;
               Pos4_Entry_Cndz_To_Exit : Bool;
               Pos4_Exit_TO_Pos4_to_Pos5 : Bool;
               Pos4_to_Pos5_TO_Pos5_Lat_Spin_Orz : Struct
                  Exe : Bool;
                  Solleva : Bool;
                  Trasla : Bool;
               END_STRUCT;
               Pos5_SpinLat_TO_Pos5_SpinLong : Bool;
            END_STRUCT;
            Ribaltatore : Struct
               MoveToPos0 : Bool;
               MoveToPos1 : Bool;
               MoveToPos2 : Bool;
               MoveToPos3 : Bool;
            END_STRUCT;
         END_STRUCT;
         P1 : Struct
            Fermi : Struct
               Rest : Bool;
               Work : Bool;
            END_STRUCT;
            Pareggiatore : Struct
               Rest : Bool;
               Work : Bool;
            END_STRUCT;
            PartMove_P1toP3_Init : Bool;
            PartMove_P1toP2_Init : Bool;
         END_STRUCT;
         P2 : Struct
            Fermi : Struct
               Rest : Bool;
               Work : Bool;
            END_STRUCT;
            Sollevatore : Struct
               EnableMove : Bool;
               Rest : Bool;
               Work : Bool;
            END_STRUCT;
            PartMove_P2toP4_Init : Bool;
         END_STRUCT;
         P3 : Struct
            Fermi : Struct
               Rest : Bool;
               Work : Bool;
            END_STRUCT;
         END_STRUCT;
         P4 : Struct
            Fermi : Struct
               Rest : Bool;
               Work : Bool;
            END_STRUCT;
            Part_Move_P2toP4_Init : Bool;
         END_STRUCT;
         P5 : Struct
            Spintore_Lat_1 : Struct
               Rest : Bool;
               Work : Bool;
            END_STRUCT;
            Spintore_Lat_2 : Struct
               Rest : Bool;
               Work : Bool;
            END_STRUCT;
            Sollevatori : Struct
               Rest : Bool;
               Work : Bool;
            END_STRUCT;
         END_STRUCT;
         Ribaltatore : Struct
            Solleva : Struct
               EnableMove : Bool;
               Rest : Bool;
               Work : Bool;
            END_STRUCT;
         END_STRUCT;
      END_STRUCT;
      Ctrl_Part_Move_P1toP2 : "Check_Part_Movement";
      Ctrl_Part_Move_P1toP3 { S7_SetPoint := 'True'} : "Check_Part_Movement";
      Ctrl_Part_Move_P2toP4 : "Check_Part_Movement";
      TON_Stop { S7_SetPoint := 'True'} : IEC_TIMER;
      TON : Struct
         BTrk_MoveP4Exit : TON_TIME;
         BTrk_MoveToP5 : TON_TIME;
         Delay_Pos1Ribalta { S7_SetPoint := 'True'} : TON_TIME;
         P1 : Struct
            Sens_Ing : Struct
               DelayOn : TON_TIME;
            END_STRUCT;
            Sens_Out : Struct
               DelayOff : TOF_TIME;
            END_STRUCT;
         END_STRUCT;
         P2 : Struct
            Sens_Ing : Struct
               DelayOn : TON_TIME;
            END_STRUCT;
            Sens_Out : Struct
               DelayOff : TOF_TIME;
            END_STRUCT;
         END_STRUCT;
         P3 : Struct
            Sens_Ing : Struct
               DelayOn : TON_TIME;
            END_STRUCT;
            Sens_Out : Struct
               DelayOff : TOF_TIME;
            END_STRUCT;
         END_STRUCT;
         P4 : Struct
            Sens_Ing : Struct
               DelayOn : TON_TIME;
            END_STRUCT;
            Sens_Out : Struct
               DelayOff : TOF_TIME;
            END_STRUCT;
         END_STRUCT;
         P1_Exit_P3 : IEC_TIMER;
         P1_Exit_P2 : IEC_TIMER;
      END_STRUCT;
      HMI : Struct
         B_ResetShiftDone : Bool;
      END_STRUCT;
      AUX : Struct
         SemiAut_Pb : Bool;
         B_ResetShiftDone : Bool;
      END_STRUCT;
      BTrk_Item : Struct   // Appoggio dati che servolo alla Stazione dopo lettura dal MES
         O_ID : DInt;
         BLean : Real;
         W_A : Real;
         H_B : Real;
         Tol_Max : Real;
         Tol_Min : Real;
         Good { ExternalAccessible := 'False'; ExternalVisible := 'False'; ExternalWritable := 'False'} : Bool;
         Bad { ExternalAccessible := 'False'; ExternalVisible := 'False'; ExternalWritable := 'False'} : Bool;
      END_STRUCT;
      PLen_Pos1 : Real;
      PLen_Pos3 : Real;
   END_VAR
   VAR_TEMP
      i : Int;   // Indice BTrk
      j : Int;   // Indice PTrk
      SensorToUse : Struct
         P1_In : Array[1..3] of Bool;
         P1_Out : Array[1..3] of Bool;   // Sensori presenza
         P2_In : Array[1..3] of Bool;
         P2_Out : Array[1..3] of Bool;   // Fotocellule
         P3_In : Array[1..3] of Bool;
         P3_Out : Array[1..3] of Bool;   // Fotocellule
         P4_In : Array[1..3] of Bool;
         P4_Out : Array[1..3] of Bool;   // Fotocellule
      END_STRUCT;
      P1 : Struct
         Cndz1_P1toP3 : Bool;
         Cndz2_P1toP3 : Bool;
      END_STRUCT;
      Trk_GetData : Struct   // Struttura dati per lettura dal MES di tutti i dati
         indx : Int;   // Se trovato tra i TODO / ENDING / OUT questo è l'indice dove sono stati prelevati i dati
         Sts : Int;   // 0 = Non Trovato; 0 = ACT; 1 = TODO; 2=ENDING; 3 = OUT
         Item : "Prod_Item_small";
      END_STRUCT;
      Sens : Struct
         P1_IngOn : Bool;
         P1_OutOn : Bool;
         P2_IngOn : Bool;
         P3_IngOn : Bool;
         P3_OutOn : Bool;
         P4_IngOn : Bool;
         P4_OutOn : Bool;
      END_STRUCT;
   END_VAR
   VAR_TEMP   // added for the SCL form of the ladder/FBD networks
      _w1 : Bool;
      _w2 : Bool;
      _w3 : Bool;
      _w4 : Bool;
      _w5 : Bool;
      _w6 : Bool;
      _w7 : Bool;
      _w8 : Bool;
      _w9 : Bool;
      _w10 : Bool;
      _w11 : Bool;
      _w12 : Bool;
      _w13 : Bool;
      _w14 : Bool;
      _w15 : Bool;
      _w16 : Bool;
      _w17 : Bool;
      _w18 : Bool;
      _w19 : Bool;
      _w20 : Bool;
      _w21 : Bool;
      _w22 : Bool;
      _w23 : Bool;
      _w24 : Bool;
      _w25 : Bool;
   END_VAR
BEGIN

REGION Network 1: °°°°°° FORZATURA PTrk °°°°°°°°°
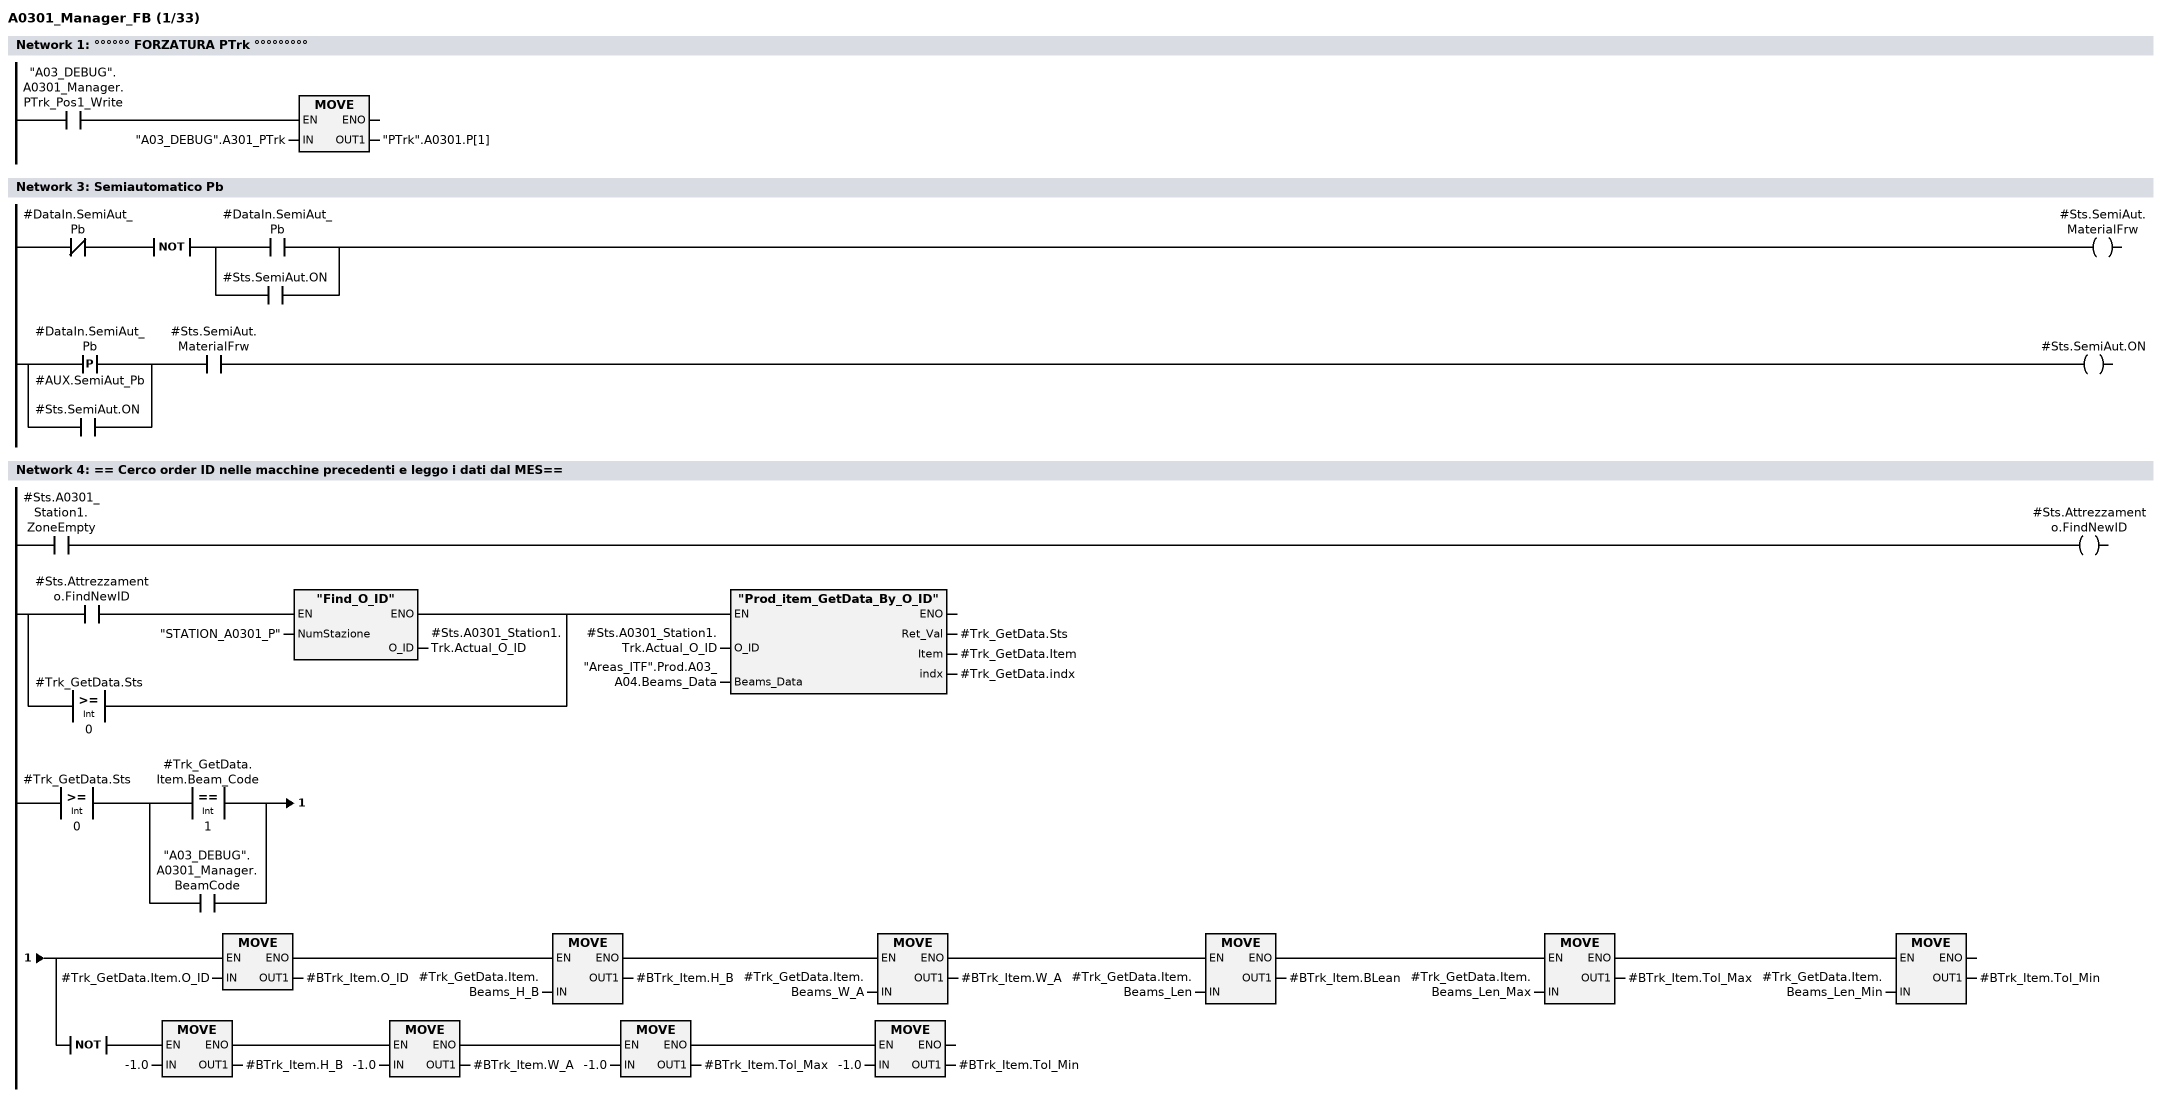
   RUNG wire#powerrail
      Contact( "A03_DEBUG".A0301_Manager.PTrk_Pos1_Write )
      Move(in := "A03_DEBUG".A301_PTrk, out1 => "PTrk".A0301.P[1])
   END_RUNG
   // the same network as SCL:
   IF "A03_DEBUG".A0301_Manager.PTrk_Pos1_Write THEN "PTrk".A0301.P[1] := "A03_DEBUG".A301_PTrk; END_IF;
END_REGION

REGION Network 2 (SCL): = Area - Rst =
   IF #AreaInterface.RstAlarms THEN
       #Alarm.WrongShiftDone := FALSE;
       #Alarm.P2toP4_NotReached:= FALSE;
       #Alarm.P1toP2_NotReached:=FALSE;
       #Alarm.P1toP3_NotReached := FALSE;
       //
       #Alarm.STOP_ControlloQualita := FALSE;
       #Alarm.STOP_FineTurno := FALSE;
       #Alarm.STOP_End_Of_Proroduction := FALSE;
   END_IF;
END_REGION

REGION Network 3: Semiautomatico Pb
   RUNG wire#powerrail
      I_Contact( #DataIn.SemiAut_Pb )
      Not()
      wire#w1
      Contact( #DataIn.SemiAut_Pb )
      wire#w2
      Coil( #Sts.SemiAut.MaterialFrw )
   END_RUNG
   RUNG wire#w1
      Contact( #Sts.SemiAut.ON )
   END_RUNG wire#w2
   RUNG wire#powerrail
      P_Contact(operand := #DataIn.SemiAut_Pb, bit := #AUX.SemiAut_Pb)
      wire#w3
      Contact( #Sts.SemiAut.MaterialFrw )
      Coil( #Sts.SemiAut.ON )
   END_RUNG
   RUNG wire#powerrail
      Contact( #Sts.SemiAut.ON )
   END_RUNG wire#w3
   // the same network as SCL:
   #Sts.SemiAut.MaterialFrw := NOT (NOT #DataIn.SemiAut_Pb) AND (#DataIn.SemiAut_Pb OR #Sts.SemiAut.ON);
   #_w1 := #DataIn.SemiAut_Pb AND NOT #AUX.SemiAut_Pb;   // rising edge of #DataIn.SemiAut_Pb
   #AUX.SemiAut_Pb := #DataIn.SemiAut_Pb;
   #Sts.SemiAut.ON := (#_w1 OR #Sts.SemiAut.ON) AND #Sts.SemiAut.MaterialFrw;
END_REGION

REGION Network 4: == Cerco order ID nelle macchine precedenti e leggo i dati dal MES==
   RUNG wire#powerrail
      Contact( #Sts.A0301_Station1.ZoneEmpty )
      Coil( #Sts.Attrezzamento.FindNewID )
   END_RUNG
   RUNG wire#powerrail
      Contact( #Sts.Attrezzamento.FindNewID )
      "Find_O_ID"(NumStazione := "STATION_A0301_P", O_ID => #Sts.A0301_Station1.Trk.Actual_O_ID)
      wire#w1
      "Prod_item_GetData_By_O_ID"(O_ID := #Sts.A0301_Station1.Trk.Actual_O_ID, Beams_Data := "Areas_ITF".Prod.A03_A04.Beams_Data, Ret_Val => #Trk_GetData.Sts, Item => #Trk_GetData.Item, indx => #Trk_GetData.indx)
   END_RUNG
   RUNG wire#powerrail
      { S7_Templates := "SrcType := Int" } GE_Contact(in1 := #Trk_GetData.Sts, in2 := 0)
   END_RUNG wire#w1
   RUNG wire#powerrail
      { S7_Templates := "SrcType := Int" } GE_Contact(in1 := #Trk_GetData.Sts, in2 := 0)
      wire#w2
      { S7_Templates := "SrcType := Int" } EQ_Contact(in1 := #Trk_GetData.Item.Beam_Code, in2 := 1)
      wire#w3
      Move(in := #Trk_GetData.Item.O_ID, out1 => #BTrk_Item.O_ID)
      Move(in := #Trk_GetData.Item.Beams_H_B, out1 => #BTrk_Item.H_B)
      Move(in := #Trk_GetData.Item.Beams_W_A, out1 => #BTrk_Item.W_A)
      Move(in := #Trk_GetData.Item.Beams_Len, out1 => #BTrk_Item.BLean)
      Move(in := #Trk_GetData.Item.Beams_Len_Max, out1 => #BTrk_Item.Tol_Max)
      Move(in := #Trk_GetData.Item.Beams_Len_Min, out1 => #BTrk_Item.Tol_Min)
   END_RUNG
   RUNG wire#w2
      Contact( "A03_DEBUG".A0301_Manager.BeamCode )
   END_RUNG wire#w3
   RUNG wire#w3
      Not()
      Move(in := -1.0, out1 => #BTrk_Item.H_B)
      Move(in := -1.0, out1 => #BTrk_Item.W_A)
      Move(in := -1.0, out1 => #BTrk_Item.Tol_Max)
      Move(in := -1.0, out1 => #BTrk_Item.Tol_Min)
   END_RUNG
   // the same network as SCL:
   #Sts.Attrezzamento.FindNewID := #Sts.A0301_Station1.ZoneEmpty;
   "Find_O_ID"(EN := #Sts.Attrezzamento.FindNewID,
               NumStazione := "STATION_A0301_P",
               O_ID => #Sts.A0301_Station1.Trk.Actual_O_ID,
               ENO => #_w1);
   IF #_w1 OR (#Trk_GetData.Sts >= 0) THEN
       #Trk_GetData.Sts := "Prod_item_GetData_By_O_ID"(O_ID := #Sts.A0301_Station1.Trk.Actual_O_ID,
                               Beams_Data := "Areas_ITF".Prod.A03_A04.Beams_Data,
                               Item => #Trk_GetData.Item,
                               indx => #Trk_GetData.indx);
   END_IF;
   #_w2 := (#Trk_GetData.Sts >= 0) AND ((#Trk_GetData.Item.Beam_Code = 1) OR "A03_DEBUG".A0301_Manager.BeamCode);
   IF #_w2 THEN
       #BTrk_Item.O_ID := #Trk_GetData.Item.O_ID;
       #BTrk_Item.H_B := #Trk_GetData.Item.Beams_H_B;
       #BTrk_Item.W_A := #Trk_GetData.Item.Beams_W_A;
       #BTrk_Item.BLean := #Trk_GetData.Item.Beams_Len;
       #BTrk_Item.Tol_Max := #Trk_GetData.Item.Beams_Len_Max;
       #BTrk_Item.Tol_Min := #Trk_GetData.Item.Beams_Len_Min;
   END_IF;
   IF NOT #_w2 THEN
       #BTrk_Item.H_B := -1.0;
       #BTrk_Item.W_A := -1.0;
       #BTrk_Item.Tol_Max := -1.0;
       #BTrk_Item.Tol_Min := -1.0;
   END_IF;
END_REGION

REGION Network 5 (SCL): == CONTROLLO TRACKING E STAZIONE PER AVANZAMENTO O_ID ==
   REGION CONTROLLO (TRK EMPTY) SU STAZIONE 1 RIBALTAMENTO A0301 
       // Controllo zona libera dai traking e sensori non in lettura su stazione A0301
       // 
       FOR #i := 1 TO "BTRK_A0301_ITEMS" DO
           IF "BTrk".A0301.B[#i].B_ID = 0 THEN
               #Sts.A0301_Station1.Trk.A0301_BTrk_Absence := TRUE;
           ELSE
               #Sts.A0301_Station1.Trk.A0301_BTrk_Absence := FALSE;
               EXIT;
           END_IF;
       END_FOR;
       //
       FOR #j := 2 TO "PTRK_A0301_ITEMS" DO
           IF "PTrk".A0301.P[#j].P_ID = 0 THEN
               #Sts.A0301_Station1.Trk.A0301_PTrk_Absence := TRUE;
           ELSE
               #Sts.A0301_Station1.Trk.A0301_PTrk_Absence := FALSE;
               EXIT;
           END_IF;
       END_FOR;

   END_REGION

   REGION CONTROLLO CHE CI SIANO LE CONDIZIONI PER MANDARE AVANTI IL NUOVO ID SU STAZIONE 1 RIBALTAMENTO A0301 (TRK EMPTY)

       // Verifica A0301 VUOTA se PTrk o BTrk assente e sensori su Stazione 1 non in lettura
       #Sts.A0301_Station1.ZoneEmpty := #Sts.A0301_Station1.Trk.A0301_PTrk_Absence AND #Sts.A0301_Station1.Trk.A0301_BTrk_Absence AND
       (NOT #Sts.P1.Fermi.Sens_Out AND
       NOT #Sts.P2.Fermi.Sens_Ing AND NOT #Sts.P1.Fermi.Sens_Out AND
       NOT #Sts.P3.Fermi.Sens_Ing AND NOT #Sts.P3.Fermi.Sens_Out AND
       NOT #Sts.P4.Fermi.Sens_Ing AND NOT #Sts.P4.Fermi.Sens_Out);


       //Se ho O_ID <> e non sono vuoto attivo avviso di attesa zona A0302 vuota
       IF (#Sts.A0301_Station1.Trk.Actual_O_ID <> #Sts.A0301_Station1.Trk.OLD_OID) OR NOT #Sts.A0301_Station1.ZoneEmpty THEN
           #Sts.A0301_Station1.Trk.Wait_A0301_Recive := TRUE;
       ELSIF (#Sts.A0301_Station1.Trk.Actual_O_ID = #Sts.A0301_Station1.Trk.OLD_OID) OR #Sts.A0301_Station1.ZoneEmpty THEN
           #Sts.A0301_Station1.Trk.Wait_A0301_Recive := FALSE;
       END_IF;

       //Se ho O_ID <> e sono vuoto aggiorno vecchio O_ID 
       IF (#Sts.A0301_Station1.Trk.Actual_O_ID <> #Sts.A0301_Station1.Trk.OLD_OID) AND #Sts.A0301_Station1.ZoneEmpty THEN
           #Sts.A0301_Station1.Trk.OLD_OID := #Sts.A0301_Station1.Trk.Actual_O_ID;
       END_IF;

   END_REGION
END_REGION

REGION Network 6 (SCL): == Compilo i dati del BTrk in base all'order ID in arrivo ==

   IF #Trk_GetData.Sts >= 0 THEN

       "BTrk".A0301.O_ID :=   #Sts.A0301_Station1.Trk.OLD_OID;
       "BTrk".A0301.Beam_Len := #BTrk_Item.BLean;
       "BTrk".A0301.Beam_W_A := #BTrk_Item.W_A;
       "BTrk".A0301.Beam_H_B := #BTrk_Item.H_B;

   ELSE
            "BTrk".A0301.O_ID := -1;
            "BTrk".A0301.Beam_Len := -1.0;
            "BTrk".A0301.Beam_W_A := -1.0;
            "BTrk".A0301.Beam_H_B := -1.0;
   END_IF;
END_REGION

REGION Network 8: <<< GESTIONE DEI SENSORI SULLE STAZIONI IN BASE ALLA LUNGHEZZA DEL PEZZO >>>
END_REGION

REGION Network 9: [P1] = Enable/Disable Sensors Pin & Controllo e Stato dei sensori ==
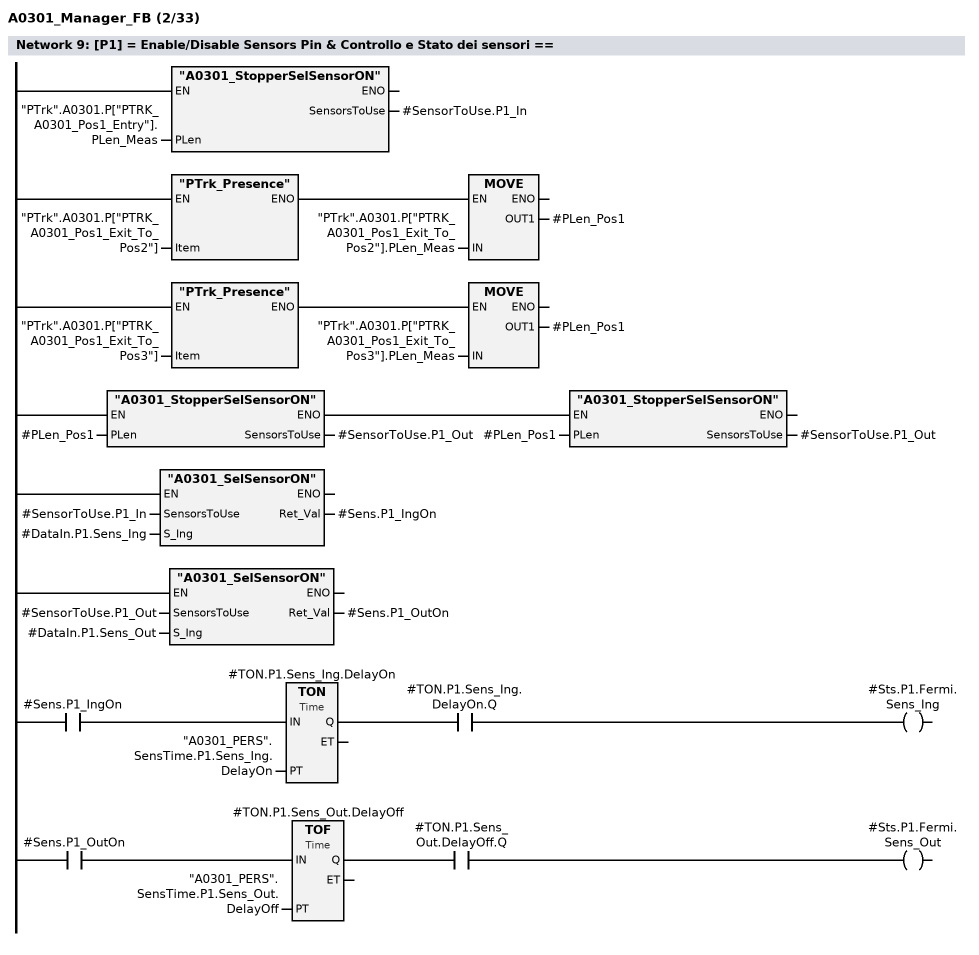
   RUNG wire#powerrail
      "A0301_StopperSelSensorON"(PLen := "PTrk".A0301.P["PTRK_A0301_Pos1_Entry"].PLen_Meas, SensorsToUse => #SensorToUse.P1_In)
   END_RUNG
   RUNG wire#powerrail
      "PTrk_Presence"(Item := "PTrk".A0301.P["PTRK_A0301_Pos1_Exit_To_Pos2"])
      Move(in := "PTrk".A0301.P["PTRK_A0301_Pos1_Exit_To_Pos2"].PLen_Meas, out1 => #PLen_Pos1)
   END_RUNG
   RUNG wire#powerrail
      "PTrk_Presence"(Item := "PTrk".A0301.P["PTRK_A0301_Pos1_Exit_To_Pos3"])
      Move(in := "PTrk".A0301.P["PTRK_A0301_Pos1_Exit_To_Pos3"].PLen_Meas, out1 => #PLen_Pos1)
   END_RUNG
   RUNG wire#powerrail
      "A0301_StopperSelSensorON"(PLen := #PLen_Pos1, SensorsToUse => #SensorToUse.P1_Out)
      "A0301_StopperSelSensorON"(PLen := #PLen_Pos1, SensorsToUse => #SensorToUse.P1_Out)
   END_RUNG
   RUNG wire#powerrail
      "A0301_SelSensorON"(SensorsToUse := #SensorToUse.P1_In, S_Ing := #DataIn.P1.Sens_Ing, Ret_Val => #Sens.P1_IngOn)
   END_RUNG
   RUNG wire#powerrail
      "A0301_SelSensorON"(SensorsToUse := #SensorToUse.P1_Out, S_Ing := #DataIn.P1.Sens_Out, Ret_Val => #Sens.P1_OutOn)
   END_RUNG
   RUNG wire#powerrail
      Contact( #Sens.P1_IngOn )
      { S7_Templates := "time_type := Time" } #TON.P1.Sens_Ing.DelayOn.TON(pt := "A0301_PERS".SensTime.P1.Sens_Ing.DelayOn, et =>)
      Contact( #TON.P1.Sens_Ing.DelayOn.Q )
      Coil( #Sts.P1.Fermi.Sens_Ing )
   END_RUNG
   RUNG wire#powerrail
      Contact( #Sens.P1_OutOn )
      { S7_Templates := "time_type := Time" } #TON.P1.Sens_Out.DelayOff.TOF(pt := "A0301_PERS".SensTime.P1.Sens_Out.DelayOff, et =>)
      Contact( #TON.P1.Sens_Out.DelayOff.Q )
      Coil( #Sts.P1.Fermi.Sens_Out )
   END_RUNG
   // the same network as SCL:
   "A0301_StopperSelSensorON"(PLen := "PTrk".A0301.P["PTRK_A0301_Pos1_Entry"].PLen_Meas,
                           SensorsToUse => #SensorToUse.P1_In);
   "PTrk_Presence"(Item := "PTrk".A0301.P["PTRK_A0301_Pos1_Exit_To_Pos2"], ENO => #_w1);
   IF #_w1 THEN #PLen_Pos1 := "PTrk".A0301.P["PTRK_A0301_Pos1_Exit_To_Pos2"].PLen_Meas; END_IF;
   "PTrk_Presence"(Item := "PTrk".A0301.P["PTRK_A0301_Pos1_Exit_To_Pos3"], ENO => #_w2);
   IF #_w2 THEN #PLen_Pos1 := "PTrk".A0301.P["PTRK_A0301_Pos1_Exit_To_Pos3"].PLen_Meas; END_IF;
   "A0301_StopperSelSensorON"(PLen := #PLen_Pos1, SensorsToUse => #SensorToUse.P1_Out, ENO => #_w3);
   IF #_w3 THEN "A0301_StopperSelSensorON"(PLen := #PLen_Pos1, SensorsToUse => #SensorToUse.P1_Out); END_IF;
   #Sens.P1_IngOn := "A0301_SelSensorON"(SensorsToUse := #SensorToUse.P1_In, S_Ing := #DataIn.P1.Sens_Ing);
   #Sens.P1_OutOn := "A0301_SelSensorON"(SensorsToUse := #SensorToUse.P1_Out, S_Ing := #DataIn.P1.Sens_Out);
   #TON.P1.Sens_Ing.DelayOn.TON(IN := #Sens.P1_IngOn, PT := "A0301_PERS".SensTime.P1.Sens_Ing.DelayOn);
   #Sts.P1.Fermi.Sens_Ing := #TON.P1.Sens_Ing.DelayOn.Q AND #TON.P1.Sens_Ing.DelayOn.Q;
   #TON.P1.Sens_Out.DelayOff.TOF(IN := #Sens.P1_OutOn, PT := "A0301_PERS".SensTime.P1.Sens_Out.DelayOff);
   #Sts.P1.Fermi.Sens_Out := #TON.P1.Sens_Out.DelayOff.Q AND #TON.P1.Sens_Out.DelayOff.Q;
END_REGION

REGION Network 10: [P2] = Enable/Disable Sensors Pin & Controllo e Stato dei sensori ==
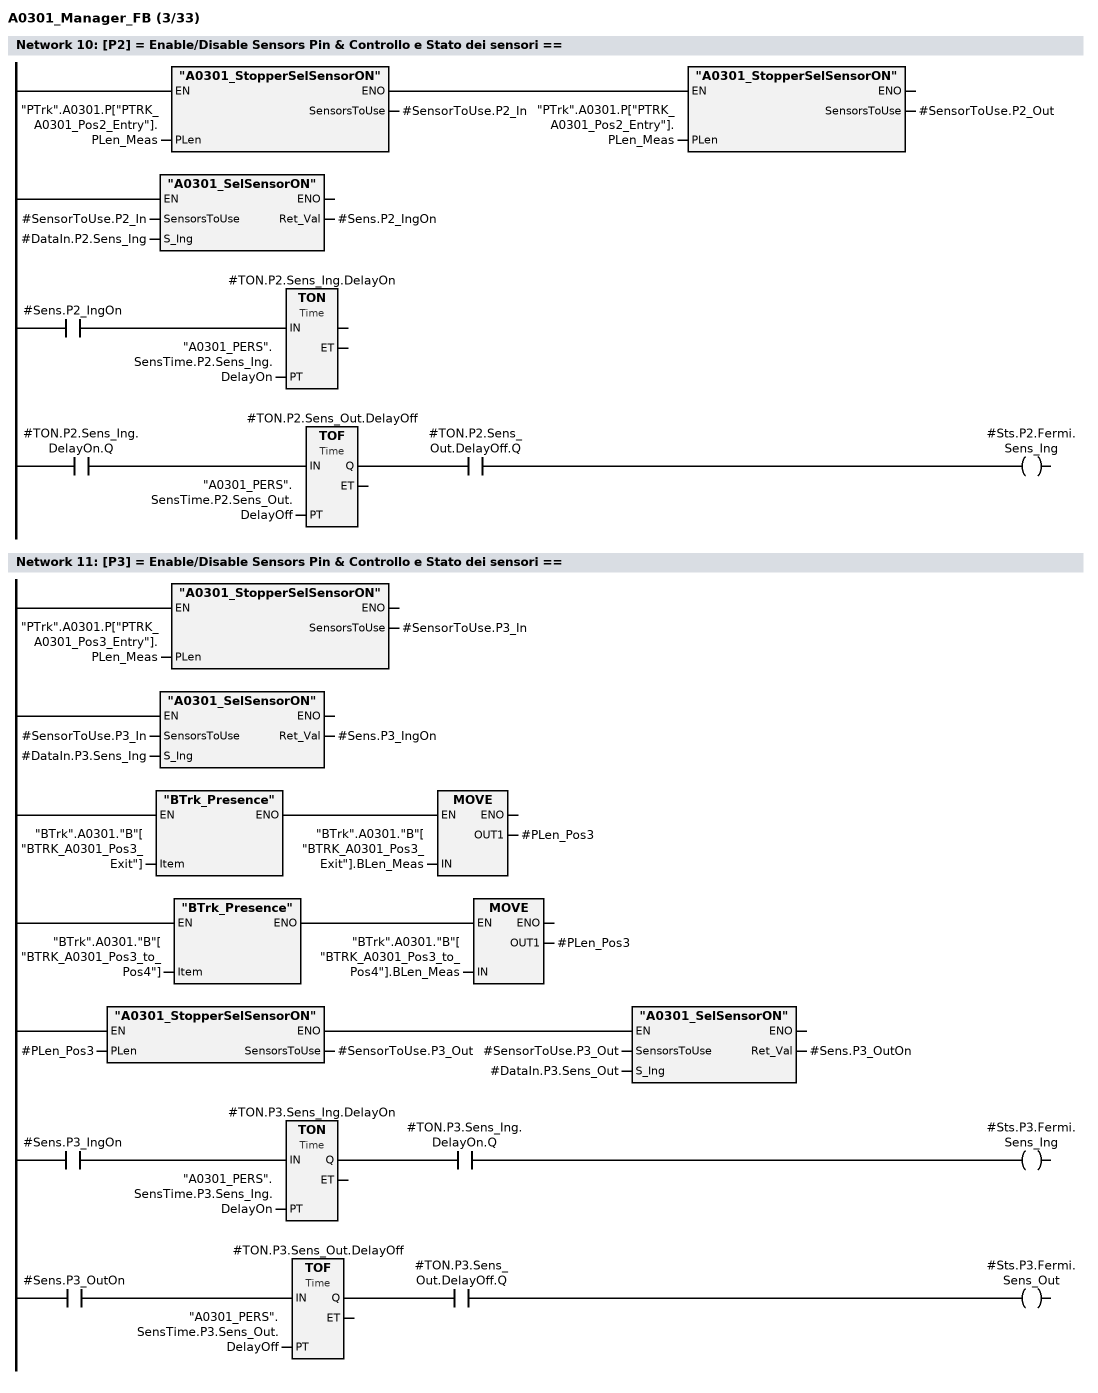
   RUNG wire#powerrail
      "A0301_StopperSelSensorON"(PLen := "PTrk".A0301.P["PTRK_A0301_Pos2_Entry"].PLen_Meas, SensorsToUse => #SensorToUse.P2_In)
      "A0301_StopperSelSensorON"(PLen := "PTrk".A0301.P["PTRK_A0301_Pos2_Entry"].PLen_Meas, SensorsToUse => #SensorToUse.P2_Out)
   END_RUNG
   RUNG wire#powerrail
      "A0301_SelSensorON"(SensorsToUse := #SensorToUse.P2_In, S_Ing := #DataIn.P2.Sens_Ing, Ret_Val => #Sens.P2_IngOn)
   END_RUNG
   RUNG wire#powerrail
      Contact( #Sens.P2_IngOn )
      { S7_Templates := "time_type := Time" } #TON.P2.Sens_Ing.DelayOn.TON(pt := "A0301_PERS".SensTime.P2.Sens_Ing.DelayOn, et =>)
   END_RUNG
   RUNG wire#powerrail
      Contact( #TON.P2.Sens_Ing.DelayOn.Q )
      { S7_Templates := "time_type := Time" } #TON.P2.Sens_Out.DelayOff.TOF(pt := "A0301_PERS".SensTime.P2.Sens_Out.DelayOff, et =>)
      Contact( #TON.P2.Sens_Out.DelayOff.Q )
      Coil( #Sts.P2.Fermi.Sens_Ing )
   END_RUNG
   // the same network as SCL:
   "A0301_StopperSelSensorON"(PLen := "PTrk".A0301.P["PTRK_A0301_Pos2_Entry"].PLen_Meas,
                           SensorsToUse => #SensorToUse.P2_In,
                           ENO => #_w1);
   IF #_w1 THEN
       "A0301_StopperSelSensorON"(PLen := "PTrk".A0301.P["PTRK_A0301_Pos2_Entry"].PLen_Meas,
                               SensorsToUse => #SensorToUse.P2_Out);
   END_IF;
   #Sens.P2_IngOn := "A0301_SelSensorON"(SensorsToUse := #SensorToUse.P2_In, S_Ing := #DataIn.P2.Sens_Ing);
   #TON.P2.Sens_Ing.DelayOn.TON(IN := #Sens.P2_IngOn, PT := "A0301_PERS".SensTime.P2.Sens_Ing.DelayOn);
   #TON.P2.Sens_Out.DelayOff.TOF(IN := #TON.P2.Sens_Ing.DelayOn.Q,
                           PT := "A0301_PERS".SensTime.P2.Sens_Out.DelayOff);
   #Sts.P2.Fermi.Sens_Ing := #TON.P2.Sens_Out.DelayOff.Q AND #TON.P2.Sens_Out.DelayOff.Q;
END_REGION

